// TwinCAT 3 PLC project Main
// ProgramVersion: 3.1.4023.0
// libraries:
//   Tc2_ModbusSrv, * (Beckhoff Automation GmbH)
//   Tc2_Standard, * (Beckhoff Automation GmbH)
//   Tc2_System, * (Beckhoff Automation GmbH)
//   Tc3_Module, * (Beckhoff Automation GmbH)
// project tree:
//   GVLs/ gvl_ha.TcGVL, gvl_mb.TcGVL, gvl_EA.TcGVL, gvl_RETAIN.TcGVL
//   / PLC1_Main.TcTTO
//   POUs/FB/ FB_Convert_2co2.TcPOU, FB_Convert_2temp.TcPOU, FB_Convert_2Zisterne.TcPOU, FB_Con_2_Value.TcPOU, FB_Count.TcPOU, FB_GarageStatus.TcPOU, FB_Heating.TcPOU, FB_Door.TcPOU, FB_Impulse_LongPress.TcPOU, FB_Light.TcPOU, FB_Impulse.TcPOU, FB_LightDimm.TcPOU, FB_LightDimmIndirectNC.TcPOU, FB_LightPIR.TcPOU, FB_ArithMittel10.TcPOU, FB_PowerSocket.TcPOU, FB_Fan.TcPOU, TP_RST.TcPOU
//   POUs/Light/ F_DimmAlgoForSwitch.TcPOU, F_LightDimmingConvertForHA.TcPOU
//   POUs/ MAIN.TcPOU, sub_Heating.TcPOU, sub_Light.TcPOU, sub_Access.TcPOU, sub_Measure.TcPOU, sub_Security.TcPOU, sub_Power.TcPOU
// real-time tasks:
//   TASK PLC1_Main: cycle T#10ms, priority 1, ADS port 350
// I/O:
//   DEVICE Gerät 1 (Beckhoff CCAT)
//   DEVICE CX8190
//     Schaltschrank (CX8190)
//   DEVICE Virtual-Ethernet
//     Werkstatt (BK9000)
// variable links:
//   Main/Main Instance <-> CX8190/Schaltschrank (CX8190)
//     PLC1_Main Inputs/gvl_EA.bID01_1 <-> ID01 (KL1104)/Channel 1/Eingang
//     PLC1_Main Inputs/gvl_EA.bID01_2 <-> ID01 (KL1104)/Channel 2/Eingang
//     PLC1_Main Inputs/gvl_EA.bID01_3 <-> ID01 (KL1104)/Channel 3/Eingang
//     PLC1_Main Inputs/gvl_EA.bID01_4 <-> ID01 (KL1104)/Channel 4/Eingang
//     PLC1_Main Inputs/gvl_EA.bID02_1 <-> ID02 (KL1104)/Channel 1/Eingang
//     PLC1_Main Inputs/gvl_EA.bID02_2 <-> ID02 (KL1104)/Channel 2/Eingang
//     PLC1_Main Inputs/gvl_EA.bID02_3 <-> ID02 (KL1104)/Channel 3/Eingang
//     PLC1_Main Inputs/gvl_EA.bID02_4 <-> ID02 (KL1104)/Channel 4/Eingang
//     PLC1_Main Inputs/gvl_EA.bID03_1 <-> ID03 (KL1104)/Channel 1/Eingang
//     PLC1_Main Inputs/gvl_EA.bID03_2 <-> ID03 (KL1104)/Channel 2/Eingang
//     PLC1_Main Inputs/gvl_EA.bID03_3 <-> ID03 (KL1104)/Channel 3/Eingang
//     PLC1_Main Inputs/gvl_EA.bID03_4 <-> ID03 (KL1104)/Channel 4/Eingang
//     PLC1_Main Inputs/gvl_EA.bID04_1 <-> ID04 (KL1104)/Channel 1/Eingang
//     PLC1_Main Inputs/gvl_EA.bID04_2 <-> ID04 (KL1104)/Channel 2/Eingang
//     PLC1_Main Inputs/gvl_EA.bID04_3 <-> ID04 (KL1104)/Channel 3/Eingang
//     PLC1_Main Inputs/gvl_EA.bID04_4 <-> ID04 (KL1104)/Channel 4/Eingang
//     PLC1_Main Inputs/gvl_EA.bID05_1 <-> ID05 (KL1104)/Channel 1/Eingang
//     PLC1_Main Inputs/gvl_EA.bID05_2 <-> ID05 (KL1104)/Channel 2/Eingang
//     PLC1_Main Inputs/gvl_EA.bID05_3 <-> ID05 (KL1104)/Channel 3/Eingang
//     PLC1_Main Inputs/gvl_EA.bID05_4 <-> ID05 (KL1104)/Channel 4/Eingang
//     PLC1_Main Inputs/gvl_EA.bID06_1 <-> ID06 (KL1104)/Channel 1/Eingang
//     PLC1_Main Inputs/gvl_EA.bID06_2 <-> ID06 (KL1104)/Channel 2/Eingang
//     PLC1_Main Inputs/gvl_EA.bID06_3 <-> ID06 (KL1104)/Channel 3/Eingang
//     PLC1_Main Inputs/gvl_EA.bID06_4 <-> ID06 (KL1104)/Channel 4/Eingang
//     PLC1_Main Inputs/gvl_EA.bID24_01_1 <-> ID24-01 (KL1104)/Channel 1/Eingang
//     PLC1_Main Inputs/gvl_EA.bID24_01_2 <-> ID24-01 (KL1104)/Channel 2/Eingang
//     PLC1_Main Inputs/gvl_EA.bID24_01_3 <-> ID24-01 (KL1104)/Channel 3/Eingang
//     PLC1_Main Inputs/gvl_EA.bID24_01_4 <-> ID24-01 (KL1104)/Channel 4/Eingang
//     PLC1_Main Inputs/gvl_EA.bID24_02_1 <-> ID24-02 (KL1104)/Channel 1/Eingang
//     PLC1_Main Inputs/gvl_EA.bID24_02_2 <-> ID24-02 (KL1104)/Channel 2/Eingang
//     PLC1_Main Inputs/gvl_EA.bID24_02_3 <-> ID24-02 (KL1104)/Channel 3/Eingang
//     PLC1_Main Inputs/gvl_EA.bID24_02_4 <-> ID24-02 (KL1104)/Channel 4/Eingang
//     PLC1_Main Inputs/gvl_EA.bID24_03_1 <-> ID24-03 (KL1104)/Channel 1/Eingang
//     PLC1_Main Inputs/gvl_EA.bID24_03_2 <-> ID24-03 (KL1104)/Channel 2/Eingang
//     PLC1_Main Inputs/gvl_EA.bID24_03_3 <-> ID24-03 (KL1104)/Channel 3/Eingang
//     PLC1_Main Inputs/gvl_EA.bID24_03_4 <-> ID24-03 (KL1104)/Channel 4/Eingang
//     PLC1_Main Inputs/gvl_EA.iIAA01_1 <-> IAA01 (KL3022)/Channel 1/Daten Ein
//     PLC1_Main Inputs/gvl_EA.iIAPT_01_1 <-> IAPT_01 (KL3214)/Channel 1/Daten Ein
//     PLC1_Main Inputs/gvl_EA.iIAV01_1 <-> IAV01 (KL3064)/Channel 1/Daten Ein
//     PLC1_Main Inputs/gvl_EA.iIAV01_2 <-> IAV01 (KL3064)/Channel 2/Daten Ein
//     PLC1_Main Inputs/gvl_EA.iIAV01_3 <-> IAV01 (KL3064)/Channel 3/Daten Ein
//     PLC1_Main Inputs/gvl_EA.iIAV01_4 <-> IAV01 (KL3064)/Channel 4/Daten Ein
//     PLC1_Main Inputs/gvl_EA.iIAV02_1 <-> IAV02 (KL3064)/Channel 1/Daten Ein
//     PLC1_Main Inputs/gvl_EA.iIAV02_2 <-> IAV02 (KL3064)/Channel 2/Daten Ein
//     PLC1_Main Inputs/gvl_EA.iIAV02_3 <-> IAV02 (KL3064)/Channel 3/Daten Ein
//     PLC1_Main Inputs/gvl_EA.iIAV02_4 <-> IAV02 (KL3064)/Channel 4/Daten Ein
//     PLC1_Main Outputs/gvl_EA.bOD01_1 <-> OD01 (KL2408)/Channel 1/Ausgang
//     PLC1_Main Outputs/gvl_EA.bOD01_2 <-> OD01 (KL2408)/Channel 2/Ausgang
//     PLC1_Main Outputs/gvl_EA.bOD01_3 <-> OD01 (KL2408)/Channel 3/Ausgang
//     PLC1_Main Outputs/gvl_EA.bOD01_4 <-> OD01 (KL2408)/Channel 4/Ausgang
//     PLC1_Main Outputs/gvl_EA.bOD01_5 <-> OD01 (KL2408)/Channel 5/Ausgang
//     PLC1_Main Outputs/gvl_EA.bOD01_6 <-> OD01 (KL2408)/Channel 6/Ausgang
//     PLC1_Main Outputs/gvl_EA.bOD01_7 <-> OD01 (KL2408)/Channel 7/Ausgang
//     PLC1_Main Outputs/gvl_EA.bOD01_8 <-> OD01 (KL2408)/Channel 8/Ausgang
//     PLC1_Main Outputs/gvl_EA.bOD02_1 <-> OD02 (KL2408)/Channel 1/Ausgang
//     PLC1_Main Outputs/gvl_EA.bOD02_2 <-> OD02 (KL2408)/Channel 2/Ausgang
//     PLC1_Main Outputs/gvl_EA.bOD02_3 <-> OD02 (KL2408)/Channel 3/Ausgang
//     PLC1_Main Outputs/gvl_EA.bOD02_4 <-> OD02 (KL2408)/Channel 4/Ausgang
//     PLC1_Main Outputs/gvl_EA.bOD02_5 <-> OD02 (KL2408)/Channel 5/Ausgang
//     PLC1_Main Outputs/gvl_EA.bOD02_6 <-> OD02 (KL2408)/Channel 6/Ausgang
//     PLC1_Main Outputs/gvl_EA.bOD02_7 <-> OD02 (KL2408)/Channel 7/Ausgang
//     PLC1_Main Outputs/gvl_EA.bOD02_8 <-> OD02 (KL2408)/Channel 8/Ausgang
//     PLC1_Main Outputs/gvl_EA.bOD03_1 <-> OD03 (KL2408)/Channel 1/Ausgang
//     PLC1_Main Outputs/gvl_EA.bOD03_2 <-> OD03 (KL2408)/Channel 2/Ausgang
//     PLC1_Main Outputs/gvl_EA.bOD03_3 <-> OD03 (KL2408)/Channel 3/Ausgang
//     PLC1_Main Outputs/gvl_EA.bOD03_4 <-> OD03 (KL2408)/Channel 4/Ausgang
//     PLC1_Main Outputs/gvl_EA.bOD03_5 <-> OD03 (KL2408)/Channel 5/Ausgang
//     PLC1_Main Outputs/gvl_EA.bOD03_6 <-> OD03 (KL2408)/Channel 6/Ausgang
//     PLC1_Main Outputs/gvl_EA.bOD03_7 <-> OD03 (KL2408)/Channel 7/Ausgang
//     PLC1_Main Outputs/gvl_EA.bOD03_8 <-> OD03 (KL2408)/Channel 8/Ausgang
//     PLC1_Main Outputs/gvl_EA.bOD04_1 <-> OD04 (KL2408)/Channel 1/Ausgang
//     PLC1_Main Outputs/gvl_EA.bOD04_2 <-> OD04 (KL2408)/Channel 2/Ausgang
//     PLC1_Main Outputs/gvl_EA.bOD04_3 <-> OD04 (KL2408)/Channel 3/Ausgang
//     PLC1_Main Outputs/gvl_EA.bOD04_4 <-> OD04 (KL2408)/Channel 4/Ausgang
//     PLC1_Main Outputs/gvl_EA.bOD04_5 <-> OD04 (KL2408)/Channel 5/Ausgang
//     PLC1_Main Outputs/gvl_EA.bOD04_6 <-> OD04 (KL2408)/Channel 6/Ausgang
//     PLC1_Main Outputs/gvl_EA.bOD04_7 <-> OD04 (KL2408)/Channel 7/Ausgang
//     PLC1_Main Outputs/gvl_EA.bOD04_8 <-> OD04 (KL2408)/Channel 8/Ausgang
//     PLC1_Main Outputs/gvl_EA.iOA01_1 <-> OA01 (KL4004)/Channel 1/Daten Aus
//     PLC1_Main Outputs/gvl_EA.iOA01_2 <-> OA01 (KL4004)/Channel 2/Daten Aus
//     PLC1_Main Outputs/gvl_EA.iOA01_3 <-> OA01 (KL4004)/Channel 3/Daten Aus
//     PLC1_Main Outputs/gvl_EA.iOA01_4 <-> OA01 (KL4004)/Channel 4/Daten Aus
//     PLC1_Main Outputs/gvl_EA.iOADim01 <-> OADim01 (KL2751)/Channel 1/Daten Aus
//     PLC1_Main Outputs/gvl_EA.iOADim02 <-> OADim02 (KL2751)/Channel 1/Daten Aus
//   Main/Main Instance <-> Virtual-Ethernet/Werkstatt (BK9000)
//     PLC1_Main Inputs/gvl_EA.bWID01_1 <-> bWID01 (KL1809)/Channel 1/Eingang
//     PLC1_Main Inputs/gvl_EA.bWID01_10 <-> bWID01 (KL1809)/Channel 10/Eingang
//     PLC1_Main Inputs/gvl_EA.bWID01_11 <-> bWID01 (KL1809)/Channel 11/Eingang
//     PLC1_Main Inputs/gvl_EA.bWID01_12 <-> bWID01 (KL1809)/Channel 12/Eingang
//     PLC1_Main Inputs/gvl_EA.bWID01_13 <-> bWID01 (KL1809)/Channel 13/Eingang
//     PLC1_Main Inputs/gvl_EA.bWID01_14 <-> bWID01 (KL1809)/Channel 14/Eingang
//     PLC1_Main Inputs/gvl_EA.bWID01_15 <-> bWID01 (KL1809)/Channel 15/Eingang
//     PLC1_Main Inputs/gvl_EA.bWID01_16 <-> bWID01 (KL1809)/Channel 16/Eingang
//     PLC1_Main Inputs/gvl_EA.bWID01_2 <-> bWID01 (KL1809)/Channel 2/Eingang
//     PLC1_Main Inputs/gvl_EA.bWID01_3 <-> bWID01 (KL1809)/Channel 3/Eingang
//     PLC1_Main Inputs/gvl_EA.bWID01_4 <-> bWID01 (KL1809)/Channel 4/Eingang
//     PLC1_Main Inputs/gvl_EA.bWID01_5 <-> bWID01 (KL1809)/Channel 5/Eingang
//     PLC1_Main Inputs/gvl_EA.bWID01_6 <-> bWID01 (KL1809)/Channel 6/Eingang
//     PLC1_Main Inputs/gvl_EA.bWID01_7 <-> bWID01 (KL1809)/Channel 7/Eingang
//     PLC1_Main Inputs/gvl_EA.bWID01_8 <-> bWID01 (KL1809)/Channel 8/Eingang
//     PLC1_Main Inputs/gvl_EA.bWID01_9 <-> bWID01 (KL1809)/Channel 9/Eingang
//     PLC1_Main Inputs/gvl_EA.bWID02_1 <-> bWID02 (KL1809)/Channel 1/Eingang
//     PLC1_Main Inputs/gvl_EA.bWID02_10 <-> bWID02 (KL1809)/Channel 10/Eingang
//     PLC1_Main Inputs/gvl_EA.bWID02_11 <-> bWID02 (KL1809)/Channel 11/Eingang
//     PLC1_Main Inputs/gvl_EA.bWID02_12 <-> bWID02 (KL1809)/Channel 12/Eingang
//     PLC1_Main Inputs/gvl_EA.bWID02_13 <-> bWID02 (KL1809)/Channel 13/Eingang
//     PLC1_Main Inputs/gvl_EA.bWID02_14 <-> bWID02 (KL1809)/Channel 14/Eingang
//     PLC1_Main Inputs/gvl_EA.bWID02_15 <-> bWID02 (KL1809)/Channel 15/Eingang
//     PLC1_Main Inputs/gvl_EA.bWID02_16 <-> bWID02 (KL1809)/Channel 16/Eingang
//     PLC1_Main Inputs/gvl_EA.bWID02_2 <-> bWID02 (KL1809)/Channel 2/Eingang
//     PLC1_Main Inputs/gvl_EA.bWID02_3 <-> bWID02 (KL1809)/Channel 3/Eingang
//     PLC1_Main Inputs/gvl_EA.bWID02_4 <-> bWID02 (KL1809)/Channel 4/Eingang
//     PLC1_Main Inputs/gvl_EA.bWID02_5 <-> bWID02 (KL1809)/Channel 5/Eingang
//     PLC1_Main Inputs/gvl_EA.bWID02_6 <-> bWID02 (KL1809)/Channel 6/Eingang
//     PLC1_Main Inputs/gvl_EA.bWID02_7 <-> bWID02 (KL1809)/Channel 7/Eingang
//     PLC1_Main Inputs/gvl_EA.bWID02_8 <-> bWID02 (KL1809)/Channel 8/Eingang
//     PLC1_Main Inputs/gvl_EA.bWID02_9 <-> bWID02 (KL1809)/Channel 9/Eingang
//     PLC1_Main Inputs/gvl_EA.iWIAA01_1 <-> IWAA01 (KL3022)/Channel 1/Daten Ein
//     PLC1_Main Inputs/gvl_EA.iWIAA01_2 <-> IWAA01 (KL3022)/Channel 2/Daten Ein
//     PLC1_Main Inputs/gvl_EA.iWIAA02_1 <-> IWAA02 (KL3054)/Channel 1/Daten Ein
//     PLC1_Main Inputs/gvl_EA.iWIAA02_2 <-> IWAA02 (KL3054)/Channel 2/Daten Ein
//     PLC1_Main Inputs/gvl_EA.iWIAA02_3 <-> IWAA02 (KL3054)/Channel 3/Daten Ein
//     PLC1_Main Inputs/gvl_EA.iWIAA02_4 <-> IWAA02 (KL3054)/Channel 4/Daten Ein
//     PLC1_Main Inputs/gvl_EA.iWIAV01_1 <-> IWAV01 (KL3064)/Channel 1/Daten Ein
//     PLC1_Main Inputs/gvl_EA.iWIAV01_2 <-> IWAV01 (KL3064)/Channel 2/Daten Ein
//     PLC1_Main Inputs/gvl_EA.iWIAV01_3 <-> IWAV01 (KL3064)/Channel 3/Daten Ein
//     PLC1_Main Inputs/gvl_EA.iWIAV01_4 <-> IWAV01 (KL3064)/Channel 4/Daten Ein
//     PLC1_Main Outputs/gvl_EA.bWOD01_1 <-> bWOD01 (KL2809)/Channel 1/Ausgang
//     PLC1_Main Outputs/gvl_EA.bWOD01_10 <-> bWOD01 (KL2809)/Channel 10/Ausgang
//     PLC1_Main Outputs/gvl_EA.bWOD01_11 <-> bWOD01 (KL2809)/Channel 11/Ausgang
//     PLC1_Main Outputs/gvl_EA.bWOD01_12 <-> bWOD01 (KL2809)/Channel 12/Ausgang
//     PLC1_Main Outputs/gvl_EA.bWOD01_13 <-> bWOD01 (KL2809)/Channel 13/Ausgang
//     PLC1_Main Outputs/gvl_EA.bWOD01_14 <-> bWOD01 (KL2809)/Channel 14/Ausgang
//     PLC1_Main Outputs/gvl_EA.bWOD01_15 <-> bWOD01 (KL2809)/Channel 15/Ausgang
//     PLC1_Main Outputs/gvl_EA.bWOD01_16 <-> bWOD01 (KL2809)/Channel 16/Ausgang
//     PLC1_Main Outputs/gvl_EA.bWOD01_2 <-> bWOD01 (KL2809)/Channel 2/Ausgang
//     PLC1_Main Outputs/gvl_EA.bWOD01_3 <-> bWOD01 (KL2809)/Channel 3/Ausgang
//     PLC1_Main Outputs/gvl_EA.bWOD01_4 <-> bWOD01 (KL2809)/Channel 4/Ausgang
//     PLC1_Main Outputs/gvl_EA.bWOD01_5 <-> bWOD01 (KL2809)/Channel 5/Ausgang
//     PLC1_Main Outputs/gvl_EA.bWOD01_6 <-> bWOD01 (KL2809)/Channel 6/Ausgang
//     PLC1_Main Outputs/gvl_EA.bWOD01_7 <-> bWOD01 (KL2809)/Channel 7/Ausgang
//     PLC1_Main Outputs/gvl_EA.bWOD01_8 <-> bWOD01 (KL2809)/Channel 8/Ausgang
//     PLC1_Main Outputs/gvl_EA.bWOD01_9 <-> bWOD01 (KL2809)/Channel 9/Ausgang
//     PLC1_Main Outputs/gvl_EA.bWOD02_1 <-> bWOD02 (KL2809)/Channel 1/Ausgang
//     PLC1_Main Outputs/gvl_EA.bWOD02_10 <-> bWOD02 (KL2809)/Channel 10/Ausgang
//     PLC1_Main Outputs/gvl_EA.bWOD02_11 <-> bWOD02 (KL2809)/Channel 11/Ausgang
//     PLC1_Main Outputs/gvl_EA.bWOD02_12 <-> bWOD02 (KL2809)/Channel 12/Ausgang
//     PLC1_Main Outputs/gvl_EA.bWOD02_13 <-> bWOD02 (KL2809)/Channel 13/Ausgang
//     PLC1_Main Outputs/gvl_EA.bWOD02_14 <-> bWOD02 (KL2809)/Channel 14/Ausgang
//     PLC1_Main Outputs/gvl_EA.bWOD02_15 <-> bWOD02 (KL2809)/Channel 15/Ausgang
//     PLC1_Main Outputs/gvl_EA.bWOD02_16 <-> bWOD02 (KL2809)/Channel 16/Ausgang
//     PLC1_Main Outputs/gvl_EA.bWOD02_2 <-> bWOD02 (KL2809)/Channel 2/Ausgang
//     PLC1_Main Outputs/gvl_EA.bWOD02_3 <-> bWOD02 (KL2809)/Channel 3/Ausgang
//     PLC1_Main Outputs/gvl_EA.bWOD02_4 <-> bWOD02 (KL2809)/Channel 4/Ausgang
//     PLC1_Main Outputs/gvl_EA.bWOD02_5 <-> bWOD02 (KL2809)/Channel 5/Ausgang
//     PLC1_Main Outputs/gvl_EA.bWOD02_6 <-> bWOD02 (KL2809)/Channel 6/Ausgang
//     PLC1_Main Outputs/gvl_EA.bWOD02_7 <-> bWOD02 (KL2809)/Channel 7/Ausgang
//     PLC1_Main Outputs/gvl_EA.bWOD02_8 <-> bWOD02 (KL2809)/Channel 8/Ausgang
//     PLC1_Main Outputs/gvl_EA.bWOD02_9 <-> bWOD02 (KL2809)/Channel 9/Ausgang

CONFIGURATION Main
    RESOURCE PLC ON TwinCAT3
        TASK PLC1_Main(INTERVAL := T#10ms, PRIORITY := 1);
        PROGRAM MAIN WITH PLC1_Main : MAIN;
    END_RESOURCE
END_CONFIGURATION

// ---- GVLs/gvl_ha.TcGVL
{attribute 'qualified_only'}
VAR_GLOBAL
	
//---------------WETTERSTATION-----------------------
	diWetterLUX			AT	%Q*:DINT;
	bWetterRAIN			AT	%Q*:BOOL;
	wWetterRAIN			AT	%Q*:WORD;
	diWetterWINDdir		AT	%Q*:DINT;
	diWetterWINDspeed	AT	%Q*:DINT;
	diWetterHUM			AT	%Q*:DINT;
	diWetterTEMP		AT	%Q*:DINT;	

END_VAR

// ---- GVLs/gvl_mb.TcGVL
{attribute 'qualified_only'}
VAR_GLOBAL
	
	Input_Coils        	: ARRAY [0..255] OF BOOL;  	//R/W BOOLS
	Input_Registers     : ARRAY [0..255] OF WORD;	//R/W 16-Bit Register
	
	Output_Coils	    : ARRAY [0..255] OF BOOL;	//Read Only BOOLS
	Output_Registers    : ARRAY [0..255] OF WORD;	//Read Only 16-Bit Register
	
END_VAR

(*-----------------------------------------------------------------------------
Output_Coils[0]		- 1000 <- Licht Küche
Output_Coils[1] 	- 1001 <- Licht Hausgang EG
Output_Coils[2] 	- 1002 <- Aussenbeleuchtung OST 		
Output_Coils[3] 	- 1003 <- Aussenbeleuchtung Haustür 	
Output_Coils[4] 	- 1004 <- Licht Technikraum
Output_Coils[5] 	- 1005 <- Licht Hobbyraum
Output_Coils[6] 	- 1006 <- Licht Werkstatt
Output_Coils[7] 	- 1007 <- Licht Esszimmertisch
Output_Coils[8] 	- 1008 <- Licht Esszimmer
Output_Coils[9] 	- 1009 <- Licht Wohnzimmer
Output_Coils[10] 	- 1010 <- Aussenbeleuchtung Balkon
Output_Coils[11] 	- 1011 <- Wohnzimmer Steckdose Uhr
Output_Coils[12] 	- 1012 <- Werkstatt Steckdose
Output_Coils[13] 	- 1013 <- Garagentor Stellung Toggle Impuls
Output_Coils[14] 	- 1014 <- Türgong Impuls
Output_Coils[15] 	- 1015 <- Vitramo Bad
Output_Coils[16] 	- 1016 <- Haustüröffner Impuls
Output_Coils[17] 	- 1017 <- Haustüröffner Dauer
Output_Coils[18] 	- 1018 <- Wohnzimmer Steckdose Fernseher
Output_Coils[19] 	- 1019 <- ENV_NoDailight
Output_Coils[20] 	- 1020 <- Wohnzimmer Steckdose Esszimmer
Output_Coils[21] 	- 1021 <- Aussensteckdose Haustür
Output_Coils[22] 	- 1022 <- Aussensteckdose Balkon
Output_Coils[23] 	- 1023 <- Strom Zisternenpumpe
Output_Coils[24] 	- 1024 <- Strom SmartMirror
Output_Coils[25] 	- 1025 <- Wohnzimmer Steckdose LED-Band
Output_Coils[26] 	- 1026 <- Lüfter Werkstatt
Output_Coils[27] 	- 1027 <- Strom Ladegeräte Werkstatt
Output_Coils[28] 	- 1028 <- Aussenbeleuchtung Treppe Süd
Output_Coils[29] 	- 1029 <- Eingang Bewegungsmelder Treppe Süd
Output_Coils[30] 	- 1030 <- Licht Garage
Output_Coils[31] 	- 1031 <- Eingang Bewegungsmelder Überdachung OST
Output_Coils[32] 	- 1032 <- Licht Aussen Hauseingang
Output_Coils[33] 	- 1033 <- Ventilator Garage
Output_Coils[34] 	- 1034 <- Türöffner  Garage Strasse
Output_Coils[35] 	- 1035 <- Türöffner Garage Haus
Output_Coils[36] 	- 1036 <- Garagentormotor Licht AN / AUS
Output_Coils[37] 	- 1037 <- Garagentor Stellung Lüften impuls
Output_Coils[38] 	- 1038 <- Garagentor Stellung AUF impuls
Output_Coils[39] 	- 1039 <- Garagentor Stellung AB impuls
Output_Coils[40] 	- 1040 <- Garagentor Stellung 1/2 impuls
Output_Coils[41] 	- 1041 <- Türöffner Werkstatt
Output_Coils[42] 	- 1042 <- Entfeuchter Werkstatt
Output_Coils[43] 	- 1043 <- Strom Ladegeräte Garage
Output_Coils[44] 	- 1044 <- Steckdose Garagendach

########################----FENSTER / TÜRKONTAKTE----################
Output_coils[200]	- 1200 <- Fenster 	EG 	BAD
Output_coils[201]	- 1201 <- Fenster 	EG 	Büro
Output_coils[202]	- 1202 <- Tür		EG	Balkontür
Output_coils[203]	- 1203 <- Fenster	UG	Keller
Output_coils[204]	- 1204 <- Fenster	UG	Technik
Output_coils[205]	- 1205 <- Fenster	UG	Hobbyraum Süd
Output_coils[206]	- 1206 <- Fenster	UG	Hobbyraum West
Output_coils[207]	- 1207 <- Tür		UG	Terassentür
Output_coils[208]	- 1208 <- Fenster	UG	Werkstatt
Output_coils[209]	- 1209 <- Tür		UG	Werkstatt
Output_coils[210]	- 1210 <- Tür		OG	Garage Strasse
Output_coils[211]	- 1211 <- Fenster	OG	Garage
Output_coils[212]	- 1212 <- Tür		OG	Garage Haus
Output_coils[213]	- 1213 <- Garagentor Status offen
Output_coils[214]	- 1214 <- Garagentor Status geschlossen
Output_coils[215]	- 1215 <- Garagentor Status Lüftung




########################----ALARM----################################
Output_coils[240]	- 1240 <- Aktiviert alle Alarmfunktionen

Output_coils[241]	- 1241 <- Aktiviert dauerhaft alle Lichter
Output_coils[242]	- 1242 <- Aktiviert dauerhaft alle Lichter INNEN
Output_coils[243]	- 1243 <- Aktiviert dauerhaft alle Lichter AUSSEN

Output_coils[244]	- 1244 <- Aktiviert dauerhaft alle Alarmsignale
Output_coils[245]	- 1245 <- Aktiviert dauerhaft alle Alarmsignale INNEN
Output_coils[246]	- 1246 <- Aktiviert dauerhaft alle Alarmsignale AUSSEN

Output_coils[247]	- 1247 <- 
Output_coils[248]	- 1248 <- 
Output_coils[249]	- 1249 <- 
Output_coils[250]	- 1250 <- 

Output_coils[251]	- 1251 <- Aktiviert Testalarm Esszimmertisch
Output_coils[252]	- 1252 <- Aktiviert Testalarm Esszimmer
Output_coils[253]	- 1253 <- Aktiviert Testalarm Wohnzimmer
Output_coils[254]	- 1254 <- Aktiviert Testalarm Balkon
Output_coils[255]	- 1255 <- 



------------------------------------------------------------------------------*)

(*-----------------------------------------------------------------------------
Output_Registers[0] 	- 2000 <- Trinkwasserverbrauch gvl_RETAIN 
Output_Registers[7] 	- 2007 <- Helligkeit Esszimmertisch
Output_Registers[8] 	- 2008 <- Helligkeit Esszimmer
Output_Registers[9] 	- 2009 <- Helligkeit Wohnzimmer
Output_Registers[10] 	- 2010 <- Helligkeit Aussenbeleuchtung Balkon
Output_Registers[11] 	- 2011 <- 
Output_Registers[12] 	- 2012 <- Zisterne Füllstand Prozent
Output_Registers[13] 	- 2013 <- Zisterne Füllstand Liter
Output_Registers[14] 	- 2014 <- Wohnzimmer Temperatur
Output_Registers[15] 	- 2015 <- Wohnzimmer Feuchtigkeit
Output_Registers[16] 	- 2016 <- Wohnzimmer CO2
Output_Registers[17] 	- 2017 <- Technikraum Temperatur
Output_Registers[18] 	- 2018 <- Technikraum Feuchtigkeit
Output_Registers[19] 	- 2019 <- Dachboden Temperatur
Output_Registers[20] 	- 2020 <- Werkstatt Temperatur
Output_Registers[21] 	- 2021 <- Werkstatt Feuchtigkeit
Output_Registers[22] 	- 2022 <- Zisternenwasserverbrauch gvl_RETAIN
Output_Registers[23] 	- 2023 <- Garage Temperatur
Output_Registers[24] 	- 2024 <- Garage Feuchtigkeit
Output_Registers[25] 	- 2025 <- Status Garagentor
Output_Registers[26] 	- 2026 <- AUSSEN Temperatur
Output_Registers[27] 	- 2027 <- AUSSEN relative Feuchte (%)
Output_Registers[28] 	- 2028 <- AUSSEN Regenmenge in mm (gvl_Retaun)
Output_Registers[29] 	- 2029 <- AUSSEN Windgeschwindigkeit m/s
Output_Registers[30] 	- 2030 <- AUSSEN Windgeschwindigkeit km/h
Output_Registers[31] 	- 2031 <- AUSSEN Windrichtung Grad




------------------------------------------------------------------------------*)

// ---- GVLs/gvl_EA.TcGVL
VAR_GLOBAL
	(* -------------------------------------------------------------------
	Beispielvariablendeklaration (%Q* = Ausgang; %I* = Eingang:
	bAusgang1			AT %Q*:BOOL;
	abAusgaenge			AT %Q*:ARRAY[0..7] OF BOOL;
	bEingang			AT %I*:BOOL;
	iSollwertAnalog  	AT %Q*:INT;
	
	Nach deklaration muss das Projekt neu Erstellt werden und die Konfiguration aktiviert werden.
	Dann kann bei den E/A Geräten die Zuordnung der Variable zum Eingang / Ausgang gemacht werden.
	
	INFO:
	im HASS muss die Variable mit .bAusgang angesprochen werden.
	---------------------------------------------------------------------- *)
	
	//----------OD01----------------------
	bOD01_1		AT	%Q*:BOOL;
	bOD01_2		AT	%Q*:BOOL;			// Lampe L2 Indirekt (Esszimmer) ACHTUNG NC
	bOD01_3		AT	%Q*:BOOL;			// Lampe L3 Indirekt (Wohnzimmer)
	bOD01_4		AT	%Q*:BOOL;			// Lampe L4 (Küche)
	bOD01_5		AT	%Q*:BOOL;			// Lampe L5 (Diele EG)
	bOD01_6		AT	%Q*:BOOL;			// Aussenlampe L6 (OST Rechts von Haustür)
	bOD01_7		AT	%Q*:BOOL;			// Aussenlampe L7 (OST Links von Haustür)
	bOD01_8		AT	%Q*:BOOL;			// Aussenlampe L8 (Süd - Ost)
	
	//----------OD02----------------------
	bOD02_1		AT	%Q*:BOOL;			// Aussenlampe L9 (Balkon Rechts)
	bOD02_2		AT	%Q*:BOOL;			// Aussenlampe L10 (Balkon Links)
	bOD02_3		AT	%Q*:BOOL;			// Tür-Gong
	bOD02_4		AT	%Q*:BOOL := TRUE;	// Steckdose S1 (Ecke Esszimmer SW)
	bOD02_5		AT	%Q*:BOOL := TRUE;	// Steckdose S2 (Balkontür Rechts Esszimmer)
	bOD02_6		AT	%Q*:BOOL;			// Steckdose S3 (Ecke Whonzimmer NW - Fernseher) ACHTUNG NC
	bOD02_7		AT	%Q*:BOOL;			// Aussensteckdose S4 (Haustür Rechts) 
	bOD02_8		AT	%Q*:BOOL;			// Aussensteckdose S5 (Balkon)

	//----------OD03----------------------
	bOD03_1		AT	%Q*:BOOL;			// Licht Hobbyraum Groß
	bOD03_2		AT	%Q*:BOOL;			// Licht Hobbyraum Klein
	bOD03_3		AT	%Q*:BOOL;			// Aussenlampe Süd-West
	bOD03_4		AT	%Q*:BOOL;			// Aussensteckdose Süd-West
	bOD03_5		AT	%Q*:BOOL;			// Licht Technikraum ACHTUNG NC
	bOD03_6		AT	%Q*:BOOL := TRUE;	// Zuleitung Strom Zisterne
	bOD03_7		AT	%Q*:BOOL;			// Aussenlampe West
	bOD03_8		AT	%Q*:BOOL;			// Aussensteckdose West

	//----------OD04----------------------
	bOD04_1		AT	%Q*:BOOL;			// Spot Küche
	bOD04_2		AT	%Q*:BOOL := TRUE;	// Zuleitung Niesche Diele EG
	bOD04_3		AT	%Q*:BOOL;			// Zuleitung Steckdose Lichtband
	bOD04_4		AT	%Q*:BOOL;			// Vitramo Bad OG
	bOD04_5		AT	%Q*:BOOL;			// Türöffner Haustür
	bOD04_6		AT	%Q*:BOOL;			//
	bOD04_7		AT	%Q*:BOOL;			//
	bOD04_8		AT	%Q*:BOOL;			//

	//----------OA01----------------------
	iOA01_1		AT	%Q*:INT;			//Wohnzimmer	0-10V Dimmer
	iOA01_2		AT	%Q*:INT;			//Esszimmer		0-10V Dimmer
	iOA01_3		AT	%Q*:INT;
	iOA01_4		AT	%Q*:INT;

	//----------ID01----------------------
	bID01_1		AT	%I*:BOOL; 			// 105 T1 (Esszimmer Indirekt)
	bID01_2		AT	%I*:BOOL; 			// 105 T2 (Wohnzimmer Indirekt)
	bID01_3		AT	%I*:BOOL; 			// 105 T3 (Deckenlampe Esstisch)
	bID01_4		AT	%I*:BOOL; 			// 104 T1 (Deckenlampe Küche)

	//----------ID02----------------------
	bID02_1		AT	%I*:BOOL;			// 105 T5 (Balkontür oben)
	bID02_2		AT	%I*:BOOL;			// 105 T6 (Balkontür unten)
	bID02_3		AT	%I*:BOOL;			// 115 T9 (Treppenabgang EG Oben)
	bID02_4		AT	%I*:BOOL;			// 115 T10 (Diele - Eingang Büro)

	//----------ID03----------------------
	bID03_1		AT	%I*:BOOL;			// 115 T11 (Diele - Eingang Esszimmer unten)
	bID03_2		AT	%I*:BOOL;			// 115 T12 (Diele - Haustür / Bad EG)
	bID03_3		AT	%I*:BOOL;			// Schalter Technikraum
	bID03_4		AT	%I*:BOOL;			// Bewegungsmelder Aussen L8 (Treppe Süd)

	//----------ID04----------------------
	bID04_1		AT	%I*:BOOL;			// Schalter Hobbyraum
	bID04_2		AT	%I*:BOOL;
	bID04_3		AT	%I*:BOOL;
	bID04_4		AT	%I*:BOOL;			// Heizungssteuerung K9 -> Vitramo Bad OG

	//----------ID05----------------------
	bID05_1		AT	%I*:BOOL;			// Taster Hausgang Garagentor
	bID05_2		AT	%I*:BOOL;			// Taster Hausgang Garagentür
	bID05_3		AT	%I*:BOOL;
	bID05_4		AT	%I*:BOOL;

	//----------ID06----------------------
	bID06_1		AT	%I*:BOOL;
	bID06_2		AT	%I*:BOOL;
	bID06_3		AT	%I*:BOOL;
	bID06_4		AT	%I*:BOOL;
	
	//----------ID24-01--------------------
	bID24_01_1		AT	%I*:BOOL;	// Türklingel Doorbird Aussen (R1)
	bID24_01_2		AT	%I*:BOOL;	// Türklingel Doorbird Innen (R1)
	bID24_01_3		AT	%I*:BOOL;	// Fensterkontakt Bad EG
	bID24_01_4		AT	%I*:BOOL;	// Fensterkontakt Büro
	
	//----------ID24-02--------------------
	bID24_02_1		AT	%I*:BOOL;	// Fensterkontakt Keller
	bID24_02_2		AT	%I*:BOOL;	// Fensterkontakt Technik
	bID24_02_3		AT	%I*:BOOL;	// Fensterkontakt Hobbyraum Süd
	bID24_02_4		AT	%I*:BOOL;	// Kontakt Terassentür UG
	
	//----------ID24-03--------------------
	bID24_03_1		AT	%I*:BOOL;	// Fensterkontakt Hobbyraum West
	bID24_03_2		AT	%I*:BOOL;	// Türkontakt Balkontür EG
	bID24_03_3		AT	%I*:BOOL;	// Wasseruhr Trinkwasser 	Impuls = 10 Liter
	bID24_03_4		AT	%I*:BOOL;	// Wasseruhr Zisterne 		Impuls = 1 Liter
	
	//----------OADim01---------------------
	iOADim01		AT	%Q*:INT;	// Dimmer Esszimmerlampe
	
	//----------OADim02---------------------
	iOADim02 		AT 	%Q*:INT;	// Dimmer Balkon
	
	//----------IAV01-----------------------
	iIAV01_1		AT	%I*:INT;	// Temperatur Wohnzimmer (°C)
	iIAV01_2		AT	%I*:INT;	// Feuchtigkeit Wohnzimmer (%)
	iIAV01_3		AT	%I*:INT;	// CO2 Wohnzimmer (ppm)
	iIAV01_4		AT	%I*:INT;	// Temperatur Technikraum (°C)
	
	//----------IAV02-----------------------
	iIAV02_1		AT	%I*:INT;	// Feuchtigkeit Technikraum (%)
	iIAV02_2		AT	%I*:INT;
	iIAV02_3		AT	%I*:INT;
	iIAV02_4		AT	%I*:INT;
	
	//----------IAA01-----------------------
	iIAA01_1		AT	%I*:INT;	//Füllstand Zisterne 4-20mA
	
	//----------IAPT_01---------------------
	iIAPT_01_1		AT	%I*:INT;	//PT Temp Bühne
	
	
	//-------------WERKSTATT-----------------------------
	
	//----------bWOD01-----------------------------------
	bWOD01_1		AT	%Q*:BOOL;				// Licht Werkstatt ACHTUNG NC
	bWOD01_2		AT	%Q*:BOOL;				// Strom Werkstatt
	bWOD01_3		AT	%Q*:BOOL;				// Entfeuchter Werkstatt
	bWOD01_4		AT	%Q*:BOOL;				// Lüfter UG
	bWOD01_5		AT	%Q*:BOOL;				// Ladegeräte Werkstatt
	bWOD01_6		AT	%Q*:BOOL;				// Garagentor Stellung Toggle
	bWOD01_7		AT	%Q*:BOOL;				// Licht Garage
	bWOD01_8		AT	%Q*:BOOL;				// Licht Überdachung
	bWOD01_9		AT	%Q*:BOOL;				// Ventilator Garage
	bWOD01_10		AT	%Q*:BOOL;				// Türöffner Garage Strasse
	bWOD01_11		AT	%Q*:BOOL;				// Türöffner Garage Haus
	bWOD01_12		AT	%Q*:BOOL;				// Garagentormotor Licht AN / AUS
	bWOD01_13		AT	%Q*:BOOL;				// Garagentor Stellung Lüften
	bWOD01_14		AT	%Q*:BOOL;				// Garagentor Stellung AUF
	bWOD01_15		AT	%Q*:BOOL;				// Garagentor Stellung AB
	bWOD01_16		AT	%Q*:BOOL;				// Garagentor Stellung 1/2
	
	//----------bWOD02-----------------------------------
	bWOD02_1		AT	%Q*:BOOL;				// Türöffner Werkstatt-Tür
	bWOD02_2		AT	%Q*:BOOL;				// Ladegeräte Garage
	bWOD02_3		AT	%Q*:BOOL;				// Steckdose Garagendach
	bWOD02_4		AT	%Q*:BOOL;				// 
	bWOD02_5		AT	%Q*:BOOL;				// 
	bWOD02_6		AT	%Q*:BOOL;				// 
	bWOD02_7		AT	%Q*:BOOL;				// 
	bWOD02_8		AT	%Q*:BOOL;				// 
	bWOD02_9		AT	%Q*:BOOL;				// 
	bWOD02_10		AT	%Q*:BOOL;				// 
	bWOD02_11		AT	%Q*:BOOL;				// 
	bWOD02_12		AT	%Q*:BOOL;				// 
	bWOD02_13		AT	%Q*:BOOL;				//
	bWOD02_14		AT	%Q*:BOOL;				// 
	bWOD02_15		AT	%Q*:BOOL;				// 
	bWOD02_16		AT	%Q*:BOOL;				//
	
	//---------bWID01-------------------------------------
	bWID01_1		AT	%I*:BOOL;				// LichtTaster Werksatt 
	bWID01_2		AT	%I*:BOOL;				// Stromschalter Werkstatt
	bWID01_3		AT	%I*:BOOL;				// Reedkontakt Werkstatttür
	bWID01_4		AT	%I*:BOOL;				// Reedkontakt Werkstattfenster
	bWID01_5		AT	%I*:BOOL;				// Taster Garage Haus
	bWID01_6		AT	%I*:BOOL;				// Taster Garage Strasse
	bWID01_7		AT	%I*:BOOL;				// Bewegungsmelder Überdachung
	bWID01_8		AT	%I*:BOOL;				// Garage Tür Strasse Input from Doorbird
	bWID01_9		AT	%I*:BOOL;				// Garage Tür Haus Input from Doorbird
	bWID01_10		AT	%I*:BOOL;				// Werkstatt Tür Input from Doorbird
	bWID01_11		AT	%I*:BOOL;				// Türkontakt Garagentür Strasse
	bWID01_12		AT	%I*:BOOL;				// Fensterkontakt Garage
	bWID01_13		AT	%I*:BOOL;				// Türkontakt Garagentür Haus
	bWID01_14		AT	%I*:BOOL;				// Lüftersignal Garagentorantrieb UAP1
	bWID01_15		AT	%I*:BOOL;				// Garagentor Status OFFEN
	bWID01_16		AT	%I*:BOOL;				// Garagentor Status GESCHLOSSEN
	
	//---------bWID02-------------------------------------
	bWID02_1		AT	%I*:BOOL;				// Licht Garagentor AN Rückmeldung
	bWID02_2		AT	%I*:BOOL;				// Regenmesser Garagendach Impuls = 0,3 mm Regen
	bWID02_3		AT	%I*:BOOL;				// Regenwächter
	bWID02_4		AT	%I*:BOOL;				// 
	bWID02_5		AT	%I*:BOOL;				// 
	bWID02_6		AT	%I*:BOOL;				// 
	bWID02_7		AT	%I*:BOOL;				// 
	bWID02_8		AT	%I*:BOOL;				// 
	bWID02_9		AT	%I*:BOOL;				// 
	bWID02_10		AT	%I*:BOOL;				// 
	bWID02_11		AT	%I*:BOOL;				// 
	bWID02_12		AT	%I*:BOOL;				// 
	bWID02_13		AT	%I*:BOOL;				// 
	bWID02_14		AT	%I*:BOOL;				// 
	bWID02_15		AT	%I*:BOOL;				// 
	bWID02_16		AT	%I*:BOOL;				// 
	
	//----------IWAV01-----------------------
	iWIAV01_1		AT	%I*:INT;	// Temperatur Werkstatt (-30 - +70 °C)
	iWIAV01_2		AT	%I*:INT;	// Feuchtigkeit Werkstatt (%)
	iWIAV01_3		AT	%I*:INT;	// Feuchtigkeit Garage (%)
	iWIAV01_4		AT	%I*:INT;	// Temperatur Garage (-30 - +70 °C)
	
	//----------IWAV01-----------------------
	iWIAA01_1		AT	%I*:INT;	// AUSSEN relative Feuchte
	iWIAA01_2		AT	%I*:INT;	// AUSSEN Temperatur (-30 - +70 °C)
	
		//----------IWAV01-----------------------
	iWIAA02_1		AT	%I*:INT;	// Windgeschwindigkeit max. 35m/s
	iWIAA02_2		AT	%I*:INT;	// Windrichtung
	iWIAA02_3		AT	%I*:INT;	// LUX aussenbereich
	iWIAA02_4		AT	%I*:INT;	//
	
END_VAR

// ---- GVLs/gvl_RETAIN.TcGVL
{attribute 'qualified_only'}
VAR_GLOBAL RETAIN
	//Brauchwassermenge verbraucht in m3
    waterConsumption : WORD;
	waterConsumptionZisterne : WORD;
	
	//Regenmenge in MM
	waterRain : WORD; 
END_VAR

// ---- POUs/MAIN.TcPOU
PROGRAM MAIN
VAR
END_VAR

//######################################################################################
//##------------------------------------ MAIN------- ---------------------------------##
//######################################################################################

sub_Light();
sub_Security();
sub_Access();
sub_Power();
sub_Measure();
sub_Heating();

END_PROGRAM

// ---- POUs/sub_Light.TcPOU
PROGRAM sub_Light
VAR
		fbLichtHausgang 		: FB_Light;
		fbLichtTechnikraum 		: FB_Light;
		fbLichtHobbyraum 		: FB_Light;
		fbLichtKueche			: FB_Light;
		fbLichtWerkstatt		: FB_Light;
		fbLichtGarage			: FB_Light;
		fbLichtEsstisch			: FB_LIghtDimm;
		fbLichtBalkon			: FB_LIghtDimm;
		fbLichtEsszimmer		: FB_LightDimmIndirectNC;
		fbLichtWohnzimmer		: FB_LightDimmIndirectNC;
		fbLichtAussenOST		: FB_LightPIR;
		fbLichtAussenHaustur	: FB_LightPIR;
		fbLichtAussenTreppeSud	: FB_LightPIR;
		fbLichtAussenEingang	: FB_LightPIR;
END_VAR

//###################################################################################
//##-----------------------------------BELEUCHTUNG---------------------------------##
//###################################################################################

//--------------------HAUSGANG EG----------------------------------
fbLichtHausgang.bInputs[0] 	:= gvl_EA.bID02_4;
fbLichtHausgang.bInputs[1] 	:= gvl_EA.bID03_1;
fbLichtHausgang.bInputs[2] 	:= gvl_EA.bID03_2;
fbLichtHausgang.bInputs[3] 	:= gvl_EA.bID02_3;

fbLichtHausgang.bInputsDoors[0] 	:= gvl_EA.bID24_01_2;

fbLichtHausgang
(
	bInputSec		:= gvl_mb.Output_Coils[242],
	bInputHA		:= gvl_mb.Output_Coils[1],
	bSunisDown		:= gvl_mb.Output_Coils[19],
	bOut 			=> gvl_EA.bOD01_5,
);
//-----------------------------------------------------------------

//--------------------KÜCHE----------------------------------------
fbLichtKueche.bInputs[0]	:= gvl_EA.bID01_4;

fbLichtKueche
(
	bInputSec	:= 	gvl_mb.Output_Coils[242],
	bInputHA	:=	gvl_mb.Output_Coils[0],
	bOut		=>	gvl_EA.bOD01_4, //Licht Küche
	bOut		=>	gvl_EA.bOD04_1,	//Spot Küche
);
//-----------------------------------------------------------------

//--------------------TECHNIKRAUM----------------------------------
fbLichtTechnikraum.bInputs[0] := gvl_EA.bID03_3;

fbLichtTechnikraum
(	
	bInputSec		:= gvl_mb.Output_Coils[242],
	bLightInv_NC	:= TRUE,
	bInputHA		:= gvl_mb.Output_Coils[4],
	bAllFlanks 		:= TRUE,
	bOut 			=> gvl_EA.bOD03_5,
);
//-----------------------------------------------------------------

//--------------------HOBBYRAUM------------------------------------
fbLichtHobbyraum.bInputs[0] := gvl_EA.bID04_1;

fbLichtHobbyraum
(	
	bInputSec		:= gvl_mb.Output_Coils[242],
	bInputHA		:= gvl_mb.Output_Coils[5],
	bAllFlanks 		:= TRUE,
	bOut 			=> gvl_EA.bOD03_1,
	bOut			=> gvl_EA.bOD03_2,
);
//-----------------------------------------------------------------

//--------------------WERKSTATT----------------------------------
fbLichtWerkstatt.bInputs[0] := gvl_EA.bWID01_1;

fbLichtWerkstatt.bInputsDoors[0] := gvl_mb.Output_coils[209];

fbLichtWerkstatt
(	
	bInputSec		:= gvl_mb.Output_Coils[242],
	bLightInv_NC	:= TRUE,
	bInputHA		:= gvl_mb.Output_Coils[6],
	bSunisDown		:= gvl_mb.Output_Coils[19],
	bOut 			=> gvl_EA.bWOD01_1,
);
//-----------------------------------------------------------------

//--------------------GARAGE----------------------------------
fbLichtGarage.bInputs[0] := gvl_EA.bWID01_5;
fbLichtGarage.bInputs[1] := gvl_EA.bWID01_6;

fbLichtGarage.bInputsDoors[0] := gvl_mb.Output_coils[210];
fbLichtGarage.bInputsDoors[1] := gvl_mb.Output_coils[212];

fbLichtGarage
(	
	bInputSec		:= gvl_mb.Output_Coils[242],
	bInputHA		:= gvl_mb.Output_Coils[30],
	bSunisDown		:= gvl_mb.Output_Coils[19],
	bOut 			=> gvl_EA.bWOD01_7,
);
//-----------------------------------------------------------------

//--------------------AUSSEN OST----------------------------------
fbLichtAussenOST
(	
	bInputSecLoop	:= gvl_mb.Output_Coils[243],
	bInputHA		:= gvl_mb.Output_Coils[2],
	bOut 			=> gvl_EA.bOD01_6,
);
//-----------------------------------------------------------------

//--------------------ESSTISCH----------------------------------
fbLichtEsstisch.bInputs[0] := gvl_EA.bID01_3;

fbLichtEsstisch
(	
	bInputSec		:= gvl_mb.Output_Coils[242],
	bInputSecTest	:= gvl_mb.Output_Coils[251],
	bInputHA		:= gvl_mb.Output_Coils[7],
	iDimmValue		:= gvl_mb.Output_Registers[7],
	iNumPress4Dimm	:= 4,
	iOut 			=> gvl_EA.iOADim01,
);
//-----------------------------------------------------------------

//--------------------BALKON----------------------------------
fbLichtBalkon.bInputs[0] := gvl_EA.bID02_2;

fbLichtBalkon
(	
	bInputSec		:= gvl_mb.Output_Coils[243],
	bInputSecTest	:= gvl_mb.Output_Coils[254],
	bInputHA		:= gvl_mb.Output_Coils[10],
	iDimmValue		:= gvl_mb.Output_Registers[10],
	bOnlyAtNight	:= TRUE,
	iNumPress4Dimm	:= 4,
	iOut 			=> gvl_EA.iOADim02,
);
//-----------------------------------------------------------------

//--------------------INDIREKTE BELEUCHTUNG ESSZIMMER--------------
fbLichtEsszimmer.bInputs[0] 	:= gvl_EA.bID01_1;
fbLichtEsszimmer.bInputs[1] 	:= gvl_EA.bID02_1;

fbLichtEsszimmer
(
	bInputSec		:= gvl_mb.Output_Coils[242],
	bInputSecTest	:= gvl_mb.Output_Coils[252],
	bInputHA		:= gvl_mb.Output_Coils[8],
	iDimmValue		:= gvl_mb.Output_Registers[8],
	iNumPress4Dimm	:= 4,
	iOut 			=> gvl_EA.iOA01_2,
	bOut			=> gvl_EA.bOD01_2,
);
//-----------------------------------------------------------------

//--------------------INDIREKTE BELEUCHTUNG WOHNZIMMER-------------
fbLichtWohnzimmer.bInputs[0] 	:= gvl_EA.bID01_2;

fbLichtWohnzimmer
(
	bInputSec		:= gvl_mb.Output_Coils[242],
	bInputSecTest	:= gvl_mb.Output_Coils[253],
	bInputHA		:= gvl_mb.Output_Coils[9],
	iDimmValue		:= gvl_mb.Output_Registers[9],
	iNumPress4Dimm	:= 4,
	iOut 			=> gvl_EA.iOA01_1,
	bOut			=> gvl_EA.bOD01_3,
);
//-----------------------------------------------------------------

//--------------------Aussenbeleuchtung Treppe Süd-------------
fbLichtAussenTreppeSud
(
	bInputSecLoop	:= gvl_mb.Output_Coils[243],
	bInputPIR		:= gvl_ea.bID03_4,
	bInputHA		:= gvl_mb.Output_Coils[28],
	tHigh			:= T#1M,
	bOut			=> gvl_ea.bOD01_8,
);

// Sync PIR to HA
gvl_mb.Output_Coils[29] := gvl_ea.bID03_4;
//-----------------------------------------------------------------

//--------------------Aussenbeleuchtung Eingang Haus-----------
fbLichtAussenEingang
(
	bInputSecLoop	:= gvl_mb.Output_Coils[243],
	bInputPIR		:= gvl_ea.bWID01_7,
	bInputHA		:= gvl_mb.Output_Coils[32],
	tHigh			:= T#1M,
	bOut			=> gvl_ea.bWOD01_8,
);

// Sync PIR to HA
gvl_mb.Output_Coils[31] := gvl_ea.bWID01_7;
//----------------------------------------------------------------

//--------------------AUSSEN HAUSTÜR----------------------------------
fbLichtAussenHaustur
(	
	bInputSecLoop	:= gvl_mb.Output_Coils[243],
	bInputPIR		:= gvl_ea.bWID01_7,
	tHigh			:= T#1M,
	bInputHA		:= gvl_mb.Output_Coils[3],
	bOut 			=> gvl_EA.bOD01_7,
);
//-----------------------------------------------------------------

END_PROGRAM

// ---- POUs/FB/FB_Light.TcPOU
FUNCTION_BLOCK FB_Light
VAR_INPUT
	bInputs			:	ARRAY[0..nSize] OF BOOL;	//Input Schalter oder Taster
	bInputsDoors	:	ARRAY[0..nSize] OF BOOL;	//Inputs for Door Contacts to put on light at Night
	bInputSec		:	BOOL := FALSE;				//Input für Security Schaltung
	bLightInv_NC	:	BOOL := FALSE;				//Ist das Licht invertiert? (NC)
	bAllFlanks		:	BOOL := FALSE;				//Alle Flanken verwenden?
	bSunIsDown		:	BOOL;
END_VAR
VAR_IN_OUT
	bInputHA		:	BOOL;						//Input (HA)
END_VAR
VAR_OUTPUT
	bOut			:	BOOL;
END_VAR
VAR CONSTANT
	nSize 			:	UINT := 5; 					//Maximale Anzahl Eingänge
END_VAR
VAR
	fbRtrig			:	ARRAY[0..nSize] OF R_TRIG;
	fbRtrigDoor		:	ARRAY[0..nSize] OF R_TRIG;
	fbFtrig			:	ARRAY[0..nSize] OF F_TRIG;
	Idx				:	UINT;
	bTrigger		:	BOOL;
END_VAR


IF bInputSec THEN	//Dauerlicht bei Security Falls
	
	IF bLightInv_NC THEN
		bOut		:= FALSE;
		bInputHA	:= TRUE;
	ELSE
		bOut		:= TRUE;
		bInputHA	:= TRUE;
	END_IF
	
ELSE	//Normale Funktion
	bTrigger := FALSE;

	//Init alle Flankentrigger und Frage diese ab
	FOR Idx := 0 TO nSize DO
	
		//Alle R_Trig
		fbRtrig[Idx](CLK:= bInputs[Idx], Q=> );
		fbRtrigDoor[Idx](CLK:= bInputsDoors[Idx], Q=> );
		
		bTrigger := bTrigger OR fbRtrig[Idx].Q;
	
		IF bAllFlanks THEN //Wenn alle Flanken
			fbFtrig[Idx](CLK:= bInputs[Idx], Q=> );
			bTrigger := bTrigger OR fbFtrig[Idx].Q;
		END_IF
	
		IF bSunIsDown THEN
			IF (NOT bOut AND NOT bLightInv_NC) OR (bOut AND bLightInv_NC) THEN 
				bTrigger := bTrigger OR fbRtrigDoor[Idx].Q;
			END_IF
		END_IF
		
	END_FOR
	

	IF bLightInv_NC THEN	//Wenn Licht Invertiert
	
		IF bInputHA THEN
			bOut	:= FALSE;
		ELSE
			bOut	:= TRUE;
		END_IF

	ELSE					//Wenn Licht nicht Invertiert 
		IF bInputHA THEN
			bOut	:= TRUE;
		ELSE
			bOut	:= FALSE;
		END_IF

	END_IF

	IF bTrigger THEN //Wenn Flanke erkannt
		bOut 			:= NOT bOut;
	
		IF bLightInv_NC THEN
			bInputHA	:= NOT bOut;
		ELSE
			bInputHa	:= bOut;
		END_IF
	END_IF
END_IF

END_FUNCTION_BLOCK

// ---- POUs/FB/FB_LightDimm.TcPOU
FUNCTION_BLOCK FB_LightDimm
VAR_INPUT
	bInputs				:	ARRAY[0..nSize] OF BOOL;	//Input Schalter oder Taster
	bInputSec			:	BOOL := FALSE;				//Input für Security Schaltung
	bInputSecTest		:	BOOL := FALSE;				//Testeingang für den Sec Modus
	bAllFlanks			:	BOOL := FALSE;				//Alle Flanken verwenden?
	bOnlyAtNight		:	BOOL := FALSE;				//Schalter funktioniert nur Nachts
	tLongPress			:	TIME := T#1000MS;			//Long Press Zeit für AUS!
	iNumPress4Dimm		:	UINT := 4;					//Reduktion der Helligkeit je Tastendruck
END_VAR
VAR_IN_OUT
	bInputHA		:	BOOL;						//Input (HA)
	iDimmValue		:	WORD;						//DimmValue Input
END_VAR
VAR_OUTPUT
	iOut			:	INT;
END_VAR
VAR CONSTANT
	nSize 			:	UINT := 5; 					//Maximale Anzahl Eingänge
END_VAR
VAR
	fbRtrig			:	ARRAY[0..nSize] OF R_TRIG;
	fbFtrig			:	ARRAY[0..nSize] OF F_TRIG;
	tonLongPress	:	ARRAY[0..nSize] OF TON;
	
	Idx				:	UINT;
	
	bSecRising		:	BOOL := TRUE;

END_VAR
VAR_TEMP
	iCountDimm		:	UINT;
	iCalcReduction	:	INT;
	
	bTrigger		:	BOOL := FALSE;
	bAllOFF			:	BOOL := FALSE;
END_VAR


IF bInputSec OR bInputSecTest THEN	//Party bei Security Falls
	
	bInputHA	:= TRUE;
	
	IF bSecRising THEN
		
		iDimmValue := iDimmValue + 5;

		IF iDimmValue = 255 THEN
			bSecRising := FALSE;
		END_IF	
	
	ELSE
	
		iDimmValue := iDimmValue - 5;

		IF iDimmValue <= 0 THEN
			bSecRising := TRUE;
		END_IF	
	
	END_IF

	
ELSE	//Normale Funktion

	//Init alle Flankentrigger und Frage diese ab
	FOR Idx := 0 TO nSize DO
	
		//Alle R_Trig
		fbRtrig[Idx](CLK:= bInputs[Idx], Q=> );
		tonLongPress[Idx](IN := bInputs[Idx], PT := tLongPress);
		
		bTrigger := bTrigger OR fbRtrig[Idx].Q;
		bAllOFF	:= bAllOFF OR tonLongPress[Idx].Q;
	
		IF bAllFlanks THEN //Wenn alle Flanken
			fbFtrig[Idx](CLK:= bInputs[Idx], Q=> );
			bTrigger := bTrigger OR fbFtrig[Idx].Q;
		END_IF
	
	END_FOR

	IF (iDimmValue > 0 OR bInputHA) AND iOut = 0 THEN		//Wenn über HA Eingeschaltet
		bInputHA	:= TRUE;
		
		IF iDimmValue = 0 THEN
			iDimmValue	:= 255;
		END_IF
	END_IF
	
	IF bOnlyAtNight THEN
		IF NOT gvl_mb.Output_Coils[19] THEN
			bTrigger	:= FALSE;
		END_IF
	END_IF
	
	IF bTrigger THEN
		
		IF iOut = 0 THEN					//Erstes Einschalten über Schalter
			bInputHA	:= TRUE;
			iDimmValue	:= 255;
		
		ELSE
			
			FOR iCountDimm := 0 TO iNumPress4Dimm DO
			
			iCalcReduction := (256 - (iCountDimm * (256 / iNumPress4Dimm)));
		
			IF iDimmValue > iCalcReduction THEN
				iDimmValue := iCalcReduction;
				EXIT;
			END_IF
		
			END_FOR
		
		END_IF
		
	END_IF

END_IF

IF bAllOFF OR bInputHA = FALSE OR iDimmValue <= 0 THEN		//Alles Ausschalten
	bInputHA	:= FALSE;
	iDimmValue	:= 0;
END_IF

iOut := F_LightDimmingConvertForHA(iDimmValue);

END_FUNCTION_BLOCK

// ---- POUs/Light/F_LightDimmingConvertForHA.TcPOU
FUNCTION F_LightDimmingConvertForHA : INT
VAR_INPUT
	iHA_DimmingValue	: INT;
END_VAR
VAR
	iConvertedValue		: INT;
END_VAR

(*---------------------------------------------------------
Converts a Dimming Value of Home Assistant (0-255) into a compatible 
Value for the Analog Output for Dimming (1-10V)
0V are not allowed as an Output. Ther must be a minimum of 1V (Dec:)
0V  =    0
1V  =  3276
10V = 32767
---------------------------------------------------------*)
IF iHA_DimmingValue = 255 THEN
	iConvertedValue := 32767;
ELSIF iHA_DimmingValue = 0 THEN
	iConvertedValue	:= 0;
ELSE
	iConvertedValue := 3276 + (iHA_DimmingValue * 115);
END_IF

F_LightDimmingConvertForHA := iConvertedValue;

END_FUNCTION

// ---- POUs/FB/FB_LightDimmIndirectNC.TcPOU
FUNCTION_BLOCK FB_LightDimmIndirectNC
VAR_INPUT
	bInputs				:	ARRAY[0..nSize] OF BOOL;	//Input Schalter oder Taster
	bInputSec			:	BOOL := FALSE;				//Input für Security Schaltung
	bInputSecTest		:	BOOL := FALSE;				//Testeingang für den Sec Modus
	bAllFlanks			:	BOOL := FALSE;				//Alle Flanken verwenden?
	tLongPress			:	TIME := T#1000MS;			//Long Press Zeit für AUS!
	tBlockTime			:	TIME := T#2000MS;			//Zeit nach Ausschalten bis wiedereinschalten
	iNumPress4Dimm		:	UINT := 4;					//Reduktion der Helligkeit je Tastendruck
END_VAR
VAR_IN_OUT
	bInputHA		:	BOOL;						//Input (HA)
	iDimmValue		:	WORD;						//DimmValue Input
END_VAR
VAR_OUTPUT
	iOut			:	INT;
	bOut			:	BOOL;
END_VAR
VAR CONSTANT
	nSize 			:	UINT := 5; 					//Maximale Anzahl Eingänge
END_VAR
VAR
	fbRtrig			:	ARRAY[0..nSize] OF R_TRIG;
	fbFtrig			:	ARRAY[0..nSize] OF F_TRIG;
	tonLongPress	:	ARRAY[0..nSize] OF TON;
	tonBlock		:	TON;
	
	Idx				:	UINT;
	
	bSecRising		:	BOOL := TRUE;
	bBlock			:	BOOL := FALSE;

END_VAR
VAR_TEMP
	iCountDimm		:	UINT;
	iCalcReduction	:	INT;
	
	bTrigger		:	BOOL := FALSE;
	bAllOFF			:	BOOL := FALSE;
END_VAR


tonBlock(IN := bBlock, PT := tBlockTime);

IF tonBlock.Q THEN
	bBlock	:= FALSE;
END_IF

IF (bInputSec OR bInputSecTest) AND NOT bBlock THEN	//Party bei Security Falls
	
	bInputHA	:= TRUE;
	bOut		:= FALSE;		// !!! NC
	
	IF bSecRising THEN
		
		iDimmValue := iDimmValue + 5;

		IF iDimmValue = 255 THEN
			bSecRising := FALSE;
		END_IF	
	
	ELSE
	
		iDimmValue := iDimmValue - 5;

		IF iDimmValue <= 0 THEN
			bSecRising := TRUE;
		END_IF	
	
	END_IF

	
ELSE	//Normale Funktion

	//Init alle Flankentrigger und Frage diese ab
	FOR Idx := 0 TO nSize DO
	
		//Alle R_Trig
		fbRtrig[Idx](CLK:= bInputs[Idx], Q=> );
		tonLongPress[Idx](IN := bInputs[Idx], PT := tLongPress);
		
		bTrigger := bTrigger OR fbRtrig[Idx].Q;
		bAllOFF	:= bAllOFF OR tonLongPress[Idx].Q;
	
		IF bAllFlanks THEN //Wenn alle Flanken
			fbFtrig[Idx](CLK:= bInputs[Idx], Q=> );
			bTrigger := bTrigger OR fbFtrig[Idx].Q;
		END_IF
	
	END_FOR

	IF (iDimmValue > 0 OR bInputHA) AND iOut = 0 AND NOT bBlock THEN		//Wenn über HA Eingeschaltet
		bInputHA	:= TRUE;
		bOut		:= FALSE;		// !!! NC
		
		IF iDimmValue = 0 THEN
			iDimmValue	:= 255;
		END_IF
	END_IF
	
	IF bTrigger AND NOT bBlock THEN
		
		IF iOut = 0 THEN					//Erstes Einschalten über Schalter
			bInputHA	:= TRUE;
			bOut		:= FALSE;			// !!! NC
			iDimmValue	:= 255;
		
		ELSE
			
			FOR iCountDimm := 0 TO iNumPress4Dimm DO
			
			iCalcReduction := (256 - (iCountDimm * (256 / iNumPress4Dimm)));
		
			IF iDimmValue > iCalcReduction THEN
				iDimmValue := iCalcReduction;
				EXIT;
			END_IF
		
			END_FOR
		
		END_IF
		
	END_IF

END_IF

IF bAllOFF OR bInputHA = FALSE OR iDimmValue <= 0 THEN		//Alles Ausschalten
	bInputHA	:= FALSE;
	bOut		:= TRUE;			// !!! NC
	iDimmValue	:= 0;
	bBlock		:= TRUE;
END_IF

iOut := F_LightDimmingConvertForHA(iDimmValue);

END_FUNCTION_BLOCK

// ---- POUs/FB/FB_LightPIR.TcPOU
FUNCTION_BLOCK FB_LightPIR
VAR_INPUT
	bInputPIR		:	BOOL;						//Input des Bewegungsmelders
	bInputSecLoop	:	BOOL := FALSE;				//Input für Security Loop
	tHigh			:	TIME;						//Zeit (ms) für High
END_VAR
VAR_IN_OUT
	bInputHA		:	BOOL;						//Input (HA)
END_VAR
VAR_OUTPUT
	bOut			:	BOOL;
END_VAR
VAR CONSTANT
	tSec			:	TIME := T#1S;
END_VAR
VAR
	fbRtrigPIR		:	R_TRIG;
	fbTrigSec		:	R_TRIG;
	
	bStateOut		:	BOOL := FALSE;

	tpPulse			:	TP_RST;
	
	tpPulseSec		:	TP;
	tofDelaySec		:	TOF;
END_VAR

// Security Loop
fbTrigSec	(CLK:= bInputPIR, Q=> );

IF bInputSecLoop THEN
	
	tpPulseSec	(IN := bStateOut, PT := tSec);
    tofDelaySec	(IN := bStateOut, PT := tSec);

	IF fbTrigSec.Q THEN
		bStateOut	:= TRUE;
	END_IF
	
	IF NOT tpPulseSec.Q THEN
		bStateOut := FALSE;
	END_IF
	
	IF NOT tofDelaySec.Q THEN
		bStateOut := TRUE;
	END_IF	

ELSIF bInputHA THEN

	bStateOut := TRUE;

ELSE

	fbRtrigPIR(CLK:= bInputPIR, Q=> );
	
	// Pulse
	tpPulse(IN := fbRtrigPIR.Q, PT := tHigh);

	IF tpPulse.Q THEN
		bStateOut	:= TRUE;
		
		//Reset Pulse bei neuer erkennung
		tpPulse.RST := fbRtrigPIR.Q;
		
	ELSE
		bStateOut 	:= FALSE;
	END_IF
	
	IF bInputPIR THEN
		bStateOut	:= TRUE;
	END_IF

END_IF

bOut		:= bStateOut;

END_FUNCTION_BLOCK

// ---- POUs/FB/TP_RST.TcPOU
FUNCTION_BLOCK TP_RST
VAR_INPUT
   IN : BOOL;
   PT : TIME;
   RST : BOOL;
END_VAR
VAR_OUTPUT
   Q : BOOL;
   ET : TIME;
END_VAR
VAR CONSTANT
   INIT : INT := 0;
   RUN_PULSE : INT := 1;
   PULSE_DONE : INT := 2;
   RESET_TIME : INT := 3;
END_VAR
VAR
   Timer : TON;
   State : INT;
END_VAR

CASE State OF
   INIT://Make sure output and timer are off
      Timer(IN:=FALSE, PT:=PT, ET=>ET);
      Q := FALSE;
      //See if user wants to start pulse
      IF IN THEN
         State := RUN_PULSE;
      END_IF
      
   RUN_PULSE://Normal pulse (output is true)
      Timer(IN:=TRUE, PT:=PT, ET=>ET);
      Q := TRUE;
      //See if timer reset requested
      IF RST THEN
         State := RESET_TIME;
      END_IF
      //See if timer expired (this overrides RST signal if timer is already done)
      IF Timer.Q THEN
         State := PULSE_DONE;
      END_IF
   
   PULSE_DONE://Pulse is done - ignore RST input
      //Keep timer TRUE to maintain ET like normal TP
      Timer(IN:=TRUE, PT:=PT, ET=>ET);
      Q := FALSE;
      //See if user shuts off timer
      IF NOT IN THEN
         State := INIT;
      END_IF
      
   RESET_TIME://User wants to extend pulse output (keep output high)
      //Reset timer (ET = 0 again)
      Timer(IN:=FALSE, PT:=PT, ET=>ET);
      Q := TRUE;
      //Watch for drop of RST - and go back to normal pulse output
      IF NOT RST THEN
         State := RUN_PULSE;
      END_IF
      
   ELSE //problem in code - reset state machine so FB doesn't freeze
      State := INIT;
      
END_CASE

END_FUNCTION_BLOCK

// ---- POUs/sub_Security.TcPOU
PROGRAM sub_Security
VAR

END_VAR

//###################################################################################
//##-----------------------------------SECURITY------------------------------------##
//###################################################################################

//--------------------Variablen Setzen----------------------------------
//ALARM GESAMT
IF gvl_mb.Output_Coils[240] THEN
	gvl_mb.Output_Coils[241] 	:= TRUE;
	gvl_mb.Output_Coils[244]	:= TRUE;
END_IF

//ALARM LICHT
IF gvl_mb.Output_Coils[241] THEN
	gvl_mb.Output_Coils[242]	:= TRUE;
	gvl_mb.Output_Coils[243]	:= TRUE;
END_IF

//ALARM NOIS
IF gvl_mb.Output_Coils[244] THEN
	gvl_mb.Output_Coils[245]	:= TRUE;
	gvl_mb.Output_Coils[246]	:= TRUE;
END_IF


//--------------------------------- INVERT Input Windows / Doors ------------------------
gvl_mb.Output_Coils[200] := NOT gvl_EA.bID24_01_3;		// Fensterkontakt Bad EG
gvl_mb.Output_Coils[201] := NOT gvl_EA.bID24_01_4;		// Fensterkontakt Büro
gvl_mb.Output_Coils[203] := NOT gvl_EA.bID24_02_1;		// Fensterkontakt Keller
gvl_mb.Output_Coils[204] := NOT gvl_EA.bID24_02_2;		// Fensterkontakt Technik
gvl_mb.Output_Coils[205] := NOT gvl_EA.bID24_02_3;		// Fensterkontakt Hobbyraum Süd
gvl_mb.Output_Coils[207] := NOT gvl_EA.bID24_02_4;		// Kontakt Terassentür UG
gvl_mb.Output_Coils[206] := NOT gvl_EA.bID24_03_1;		// Fensterkontakt Hobbyraum West
gvl_mb.Output_Coils[202] := NOT gvl_EA.bID24_03_2;		// Kontakt Balkontür
gvl_mb.Output_Coils[209] := NOT gvl_EA.bWID01_3;		// Reedkontakt Werkstatttür
gvl_mb.Output_Coils[208] := NOT gvl_EA.bWID01_4;		// Reedkontakt Werkstattfenster
gvl_mb.Output_coils[210] :=	NOT gvl_EA.bWID01_11; 		// TüR		OG	Garage Strasse
gvl_mb.Output_coils[211] :=	NOT gvl_EA.bWID01_12; 		// Fenster	OG	Garage
gvl_mb.Output_Coils[212] :=	NOT gvl_EA.bWID01_13; 		// TüR		OG	Garage Haus

gvl_mb.Output_coils[213] :=	gvl_EA.bWID01_15; 			// Garagentor offen
gvl_mb.Output_coils[214] := gvl_EA.bWID01_16; 			// Garagentor geschlossen
gvl_mb.Output_Coils[215] := gvl_EA.bWID01_14; 			// Garagentor Lüftung

END_PROGRAM

// ---- POUs/sub_Access.TcPOU
PROGRAM sub_Access
VAR
	
	bGarageStellungLueften	    : BOOL;
	bGarageStellungLueftenTemp	: BOOL;

	fbTuerGong			:	FB_Impulse;
	fbGaragentorToggle	:	FB_Impulse_LongPress;
	fbGaragentorAuf		:	FB_Impulse;
	fbGaragentorAb		:	FB_Impulse;
	fbGaragentorHalb	:	FB_Impulse;
	fbGaragentorLueften	:	FB_Impulse;
	fbgaragentorStatus	:	FB_GarageStatus;
	
	fbTuerGarageHaus	:	FB_Door;
	fbTuerGarageStrasse	:	FB_Door;
	fbTuerWerkstatt		:	FB_Door;
	fbTuerHaus			:	FB_Door;
	
END_VAR

//###################################################################################
//##-----------------------------------ACCESS--------------------------------------##
//###################################################################################

bGarageStellungLueften := FALSE;

//--------------------TürGong----------------------------------
fbTuerGong.bInputs[0]	:= gvl_EA.bID24_01_1;

fbTuerGong(
	bR_Trig			:= TRUE,
	bInputSecLoop	:= gvl_mb.Output_Coils[245],
	bInputHA		:= gvl_mb.Output_Coils[14],
	tHigh			:= T#500MS,
	bOut			=> gvl_EA.bOD02_3
);
//-------------------------------------------------------------

//--------------------Garagentor Stellung Auf----------------------------------
fbGaragentorAuf(
	bR_Trig			:= TRUE,
	bInputHA		:= gvl_mb.Output_Coils[38],
	tHigh			:= T#500MS,
	bOut			=> gvl_EA.bWOD01_14
);
//-------------------------------------------------------------

//--------------------Garagentor Stellung Ab----------------------------------
fbGaragentorAb(
	bR_Trig			:= TRUE,
	bInputHA		:= gvl_mb.Output_Coils[39],
	tHigh			:= T#500MS,
	bOut			=> gvl_EA.bWOD01_15
);
//-------------------------------------------------------------

//--------------------Garagentor Stellung Halb----------------------------------
fbGaragentorHalb(
	bR_Trig			:= TRUE,
	bInputHA		:= gvl_mb.Output_Coils[40],
	tHigh			:= T#500MS,
	bOut			=> gvl_EA.bWOD01_16
);
//-------------------------------------------------------------

//--------------------Garagentor Stellung Lüften----------------------------------
fbGaragentorLueften(
	bR_Trig			:= TRUE,
	bInputHA		:= gvl_mb.Output_Coils[37],
	tHigh			:= T#500MS,
	bOut			=> bGarageStellungLueftenTemp
);

bGarageStellungLueften := bGarageStellungLueften OR bGarageStellungLueftenTemp; 
//-------------------------------------------------------------

//--------------------Garagentor Stellung Toggle----------------------------------
fbGaragentorToggle(
	bInput			:= gvl_EA.bID05_1,
	bInputHA		:= gvl_mb.Output_Coils[13],
	tHigh			:= T#500MS,
	tLongPress		:= T#1S,
	bOut			=> gvl_EA.bWOD01_6,
	bOutLong		=> bGarageStellungLueftenTemp
);

bGarageStellungLueften := bGarageStellungLueften OR bGarageStellungLueftenTemp; 
//-------------------------------------------------------------

//--------------------Garagentor Status----------------------------------
fbGaragentorStatus(
	bInputOpened	:= gvl_EA.bWID01_15,
	bInputClosed	:= gvl_EA.bWID01_16,
	bInputAir		:= gvl_EA.bWID01_14,
	iOut			=> gvl_mb.Output_Registers[25]
);
//-------------------------------------------------------------

//--------------------Türöffner Garagentür Haus----------------------------------
fbTuerGarageHaus(
	bInput			:= gvl_EA.bWID01_9,
	bInputSwitch	:= gvl_EA.bID05_2,
	bInputHA		:= gvl_mb.Output_Coils[35],
	tPulse			:= T#3S,
	tPulseSwitch	:= T#10S,
	bOut			=> gvl_EA.bWOD01_11
);
//-------------------------------------------------------------

//--------------------Türöffner Garagentür Strasse----------------------------------
fbTuerGarageStrasse(
	bInput			:= gvl_EA.bWID01_8,
	bInputHA		:= gvl_mb.Output_Coils[34],
	tPulse			:= T#3S,
	bOut			=> gvl_EA.bWOD01_10
);
//-------------------------------------------------------------

//--------------------Türöffner Werkstatt----------------------------------
fbTuerWerkstatt(
	bInput			:= gvl_EA.bWID01_10,
	bInputHA		:= gvl_mb.Output_Coils[41],
	tPulse			:= T#3S,
	bOut			=> gvl_EA.bWOD02_1
);
//-------------------------------------------------------------

//--------------------Türöffner Haustür----------------------------------
fbTuerHaus(
	bInput			:= gvl_EA.bID24_01_2,
	bInputHA		:= gvl_mb.Output_Coils[16],
	bInputPerm		:= gvl_mb.Output_Coils[17],
	tPulse			:= T#5S,
	bOut			=> gvl_EA.bOD04_5
);
//-------------------------------------------------------------


gvl_EA.bWOD01_13 := bGarageStellungLueften;

END_PROGRAM

// ---- POUs/FB/FB_Impulse.TcPOU
FUNCTION_BLOCK FB_Impulse
VAR_INPUT
	bInputs			:	ARRAY[0..nSize] OF BOOL;	//Input Schalter oder Taster
	bInputSecLoop	:	BOOL := FALSE;				//Input für Security Loop
	bR_Trig			:	BOOL := TRUE;				//Steigende Flanke? Wenn FALSE = Fallend
	tHigh			:	TIME;						//Zeit (ms) für High
	tDelay			:	TIME := T#0MS;				//Verzögerungszeit (ms) zwischen den Impulsen									
END_VAR
VAR_OUTPUT
	bOut			:	BOOL;
END_VAR
VAR_IN_OUT
	bInputHA		:	BOOL;
END_VAR
VAR CONSTANT
	nSize 			:	UINT := 5; 					//Maximale Anzahl Eingänge
END_VAR
VAR
	fbRtrig			:	ARRAY[0..nSize] OF R_TRIG;
	fbFtrig			:	ARRAY[0..nSize] OF F_TRIG;
	
	fbRtrigInit		:	R_TRIG;
	
	Idx				:	UINT;
	bTrigger		:	BOOL;
	
	tpPulse			:	TP;
	tofDelay		:	TOF;
	
END_VAR
VAR_TEMP

END_VAR



//--------------------------------------Notfall Toggle
fbRtrigInit(CLK:= bInputSecLoop, Q=> );
tpPulse(IN := bOut, PT := tHigh);
tofDelay(IN := bOut, PT := tHigh);

IF bInputSecLoop THEN
		
	IF fbRtrigInit.Q THEN
		bOut	:= TRUE;
	END_IF
	
	IF NOT tpPulse.Q THEN
		bOut := FALSE;
	END_IF
	
	IF NOT tofDelay.Q THEN
		bOut := TRUE;
	END_IF	
	
ELSE //----------------------------------Normaler Impuls
	bTrigger 	:= FALSE;

	//Init alle Flankentrigger und Frage diese ab
	FOR Idx := 0 TO nSize DO
	
		IF bR_Trig THEN
		
			fbRtrig[Idx](CLK:= bInputs[Idx], Q=> );
			bTrigger := bTrigger OR fbRtrig[Idx].Q;
	
		ELSE
	
			fbFtrig[Idx](CLK:= bInputs[Idx], Q=> );
			bTrigger := bTrigger OR fbFtrig[Idx].Q;
	
		END_IF
	
	END_FOR
	
	bTrigger := bTrigger OR bInputHA;
	
	IF NOT tofDelay.Q THEN
		tpPulse(IN := bTrigger, PT := tHigh);
	END_IF

	IF tpPulse.Q THEN
		bOut 		:= TRUE;
		bInputHA 	:= TRUE;
	ELSE
		bOut 		:= FALSE;
		bInputHA	:= FALSE;
		tofDelay(IN := bOut, PT := tDelay);
	END_IF
	
END_IF

END_FUNCTION_BLOCK

// ---- POUs/FB/FB_Impulse_LongPress.TcPOU
FUNCTION_BLOCK FB_Impulse_LongPress
VAR_INPUT
	bInput			:	BOOL;	//Input Schalter oder Taster
	tHigh			:	TIME;						//Zeit (ms) für High
	tLongPress		:	TIME;							
END_VAR
VAR_OUTPUT
	bOut			:	BOOL;
	bOutLong		:	BOOL;
END_VAR
VAR_IN_OUT
	bInputHA		:	BOOL;
END_VAR
VAR CONSTANT
END_VAR
VAR
	fbFtrig			:	F_TRIG;
	bTrigger		:	BOOL;
	bOutTrig		:	BOOL;
	
	tpPulse			:	TP;
	tonLongPress	:	TON;
	
END_VAR
VAR_TEMP

END_VAR


tpPulse		 (IN := bOutTrig, PT := tHigh);
tonLongPress (IN := bInput, PT := tLongPress);

bTrigger 	:= FALSE;
		
fbFtrig(CLK:= bInput, Q=> );

//Normale Tastendruck
bTrigger := bTrigger OR fbFtrig.Q;

//Signal über HA
bTrigger := bTrigger OR bInputHA;

//Wenn normaler Tastendruck und Impuls noch nicht abgelaufen
IF (tpPulse.Q AND NOT bInput) OR bTrigger THEN
	bOut 		:= TRUE;
	bInputHA	:= FALSE;
//Wenn langer Tastendruck
ELSIF tonLongPress.Q OR (tpPulse.Q AND bInput) THEN
	bOutLong	:= TRUE;

//Wenn nichts
ELSE
	bOut 		:= FALSE;
	bOutLong	:= FALSE;
	bInputHA	:= FALSE;
	
	bOutTrig	:= FALSE;
END_IF
	
bOutTrig := bOut OR bOutLong;

END_FUNCTION_BLOCK

// ---- POUs/FB/FB_GarageStatus.TcPOU
FUNCTION_BLOCK FB_GarageStatus
VAR_INPUT
	bInputOpened	:	BOOL;
	bInputClosed	:	BOOL;
	bInputAir		:	BOOL;

END_VAR
VAR_OUTPUT
	iOut			:	INT;
END_VAR
VAR_IN_OUT
END_VAR
VAR CONSTANT
END_VAR
VAR
	fbRtrig			:	R_TRIG;
	fbRtrigSwitch	:	R_TRIG;
	fbRtrigHA		:	R_TRIG;
	
	tpPulse			:	TP;
	tpPulseSwitch	:	TP;
		
	bTrigger		:	BOOL;
	

	
	bInputOpenedAND: INT;
END_VAR
VAR_TEMP

END_VAR


IF bInputOpened AND NOT bInputClosed AND NOT bInputAir THEN
	//Geöffnet
	iOut := 3;
ELSIF NOT bInputOpened AND bInputClosed AND NOT bInputAir THEN
	//Geschlossen
	iOut := 2;
ELSIF NOT bInputOpened AND NOT bInputClosed AND bInputAir THEN
	//Lüftungstellung
	iOut := 1;
ELSE
	// Teilgeöffnet
	iOut := 0;
END_IF

END_FUNCTION_BLOCK

// ---- POUs/FB/FB_Door.TcPOU
FUNCTION_BLOCK FB_Door
VAR_INPUT
	bInput			:	BOOL;	// Input über ein System
	bInputSwitch	:	BOOL;	// Input über einen Taster
	bInputPerm		:	BOOL;	// Input für dauerhaftes öffnen
	
	tPulse			:	TIME := T#5S;	//Zeit für High bei System oder HomeAssistant
	tPulseSwitch	:	TIME := tPulse;	//Zeit für High bei Schalter 
END_VAR
VAR_OUTPUT
	bOut			:	BOOL;
END_VAR
VAR_IN_OUT
	bInputHA		:	BOOL;	// Input über Home Assistant Taster
END_VAR
VAR CONSTANT
END_VAR
VAR
	fbRtrig			:	R_TRIG;
	fbRtrigSwitch	:	R_TRIG;
	fbRtrigHA		:	R_TRIG;
	
	tpPulse			:	TP;
	tpPulseSwitch	:	TP;
		
	bTrigger		:	BOOL;
	

	
END_VAR
VAR_TEMP

END_VAR

IF bInputPerm THEN
	
	bOut := TRUE;
	
ELSE

	bTrigger 	:= FALSE;

	fbRtrig(CLK:= bInput, Q=> );
	fbRtrigSwitch(CLK:= bInputSwitch, Q=> );
	fbRtrigHA(CLK:= bInputHA, Q=> );

	bTrigger := bTrigger OR fbRtrig.Q OR fbRtrigHA.Q;
	
	tpPulse(IN := bTrigger, PT := tPulse);
	tpPulseSwitch(IN := fbRtrigSwitch.Q, PT := tPulseSwitch);

	IF tpPulse.Q OR tpPulseSwitch.Q THEN
		bOut 		:= TRUE;
	ELSE
		bOut 		:= FALSE;
		bInputHA	:= FALSE;
	END_IF
	
END_IF

END_FUNCTION_BLOCK

// ---- POUs/sub_Power.TcPOU
PROGRAM sub_Power
VAR
		fbPowerWerkstatt		:	FB_PowerSocket;
		fbPowerFernseher		:	FB_PowerSocket;
		fbPowerUhr				:	FB_PowerSocket;
		fbPowerEsszimmer		:	FB_PowerSocket;
		fbPowerAussenHaustur	:	FB_PowerSocket;
		fbPowerAussenBalkon		:	FB_PowerSocket;
		fbPowerZisterne			:	FB_PowerSocket;
		fbPowerSmartMirror		:	FB_PowerSocket;
		fbPowerLEDBandWohn		:	FB_PowerSocket;
		fbPowerLadeWerkstatt	:	FB_PowerSocket;
		fbPowerLadeGarage		:	FB_PowerSocket;
		fbPowerGaragenDach		:	FB_PowerSocket;
		
END_VAR

//###################################################################################
//##-----------------------------------POWER---------------------------------------##
//###################################################################################

//--------------------WERKSTATT STECKDOSE----------------------------------
fbPowerWerkstatt.bInputs[0] 	:= gvl_EA.bWID01_2;

fbPowerWerkstatt
(
	bPowerInv_NC	:=	TRUE,
	bInputHA		:=	gvl_mb.Output_Coils[12]	,
	bOut			=>	gvl_EA.bWOD01_2,
);
//-------------------------------------------------------------------------

//--------------------FERNSEHER STECKDOSE----------------------------------
fbPowerFernseher
(
	bPowerInv_NC	:=	TRUE,
	bInputHA		:=	gvl_mb.Output_Coils[18],
	bOut			=>	gvl_EA.bOD02_6,
);
//-------------------------------------------------------------------------

//--------------------UHR STECKDOSE----------------------------------
fbPowerUhr
(
	bInputHA		:=	gvl_mb.Output_Coils[11],
	bOut			=>	gvl_EA.bOD02_5,
);
//-------------------------------------------------------------------------

//--------------------ESSZIMMER STECKDOSE----------------------------------
fbPowerEsszimmer
(
	bInputHA		:=	gvl_mb.Output_Coils[20],
	bOut			=>	gvl_EA.bOD02_4,
);
//-------------------------------------------------------------------------

//--------------------HAUSTÜR AUSSENSTECKDOSE----------------------------------
fbPowerAussenHaustur
(
	bInputHA		:=	gvl_mb.Output_Coils[21],
	bOut			=>	gvl_EA.bOD02_7,
);
//-------------------------------------------------------------------------

//--------------------BALKON AUSSENSTECKDOSE----------------------------------
fbPowerAussenBalkon
(
	bInputHA		:=	gvl_mb.Output_Coils[22],
	bOut			=>	gvl_EA.bOD02_8,
);
//-------------------------------------------------------------------------

//--------------------STROM ZISTERNE----------------------------------
fbPowerZisterne
(
	bInputHA		:=	gvl_mb.Output_Coils[23],
	bOut			=>	gvl_EA.bOD03_6,
);
//-------------------------------------------------------------------------

//--------------------STROM SMARTMIRROR----------------------------------
fbPowerSmartMirror
(
	bInputHA		:=	gvl_mb.Output_Coils[24],
	bOut			=>	gvl_EA.bOD04_2,
);
//-------------------------------------------------------------------------

//--------------------LED-BAND WOHNZIMMER STECKDOSE-------------------------------
fbPowerLEDBandWohn
(
	bInputHA		:=	gvl_mb.Output_Coils[25],
	bOut			=>	gvl_EA.bOD04_3,
);
//-------------------------------------------------------------------------

//--------------------LADEGERÄTE WERKSTATT----------------------------------
fbPowerLadeWerkstatt
(
	bInputHA		:=	gvl_mb.Output_Coils[27],
	bOut			=>	gvl_EA.bWOD01_5,
);
//-------------------------------------------------------------------------

//--------------------LADEGERÄTE GARAGE----------------------------------
fbPowerLadeGarage
(
	bInputHA		:=	gvl_mb.Output_Coils[43],
	bOut			=>	gvl_EA.bWOD02_2,
);
//-------------------------------------------------------------------------

//--------------------STECKDOSE GARAGENDACH----------------------------------
fbPowerGaragenDach
(
	bInputHA		:=	gvl_mb.Output_Coils[44],
	bOut			=>	gvl_EA.bWOD02_3,
);
//-------------------------------------------------------------------------

END_PROGRAM

// ---- POUs/FB/FB_PowerSocket.TcPOU
FUNCTION_BLOCK FB_PowerSocket
VAR_INPUT
	bInputs			:	ARRAY[0..nSize] OF BOOL;	//Input Schalter oder Taster
	bPowerInv_NC	:	BOOL := FALSE;				//Ist die Schaltung invertiert? (NC)
	bAllFlanks		:	BOOL := FALSE;				//Alle Flanken verwenden?
END_VAR
VAR_IN_OUT
	bInputHA		:	BOOL;						//Input (HA)
END_VAR
VAR_OUTPUT
	bOut			:	BOOL;
END_VAR
VAR CONSTANT
	nSize 			:	UINT := 5; 					//Maximale Anzahl Eingänge
END_VAR
VAR
	fbRtrig			:	ARRAY[0..nSize] OF R_TRIG;
	fbFtrig			:	ARRAY[0..nSize] OF F_TRIG;
	Idx				:	UINT;
	bTrigger		:	BOOL;
END_VAR


bTrigger := FALSE;

//Init alle Flankentrigger und Frage diese ab
FOR Idx := 0 TO nSize DO
	
	//Alle R_Trig
	fbRtrig[Idx](CLK:= bInputs[Idx], Q=> );
	bTrigger := bTrigger OR fbRtrig[Idx].Q;
	
	IF bAllFlanks THEN //Wenn alle Flanken
		fbFtrig[Idx](CLK:= bInputs[Idx], Q=> );
		bTrigger := bTrigger OR fbFtrig[Idx].Q;
	END_IF
	
END_FOR

IF bPowerInv_NC THEN	//Wenn Schaltung Invertiert
	
	IF bInputHA THEN
		bOut	:= FALSE;
	ELSE
		bOut	:= TRUE;
	END_IF

ELSE					//Wenn Licht nicht Invertiert 
	IF bInputHA THEN
		bOut	:= TRUE;
	ELSE
		bOut	:= FALSE;
	END_IF

END_IF

IF bTrigger THEN //Wenn Flanke erkannt
	
	bOut 			:= NOT bOut;
	
	IF bPowerInv_NC THEN
		bInputHA	:= NOT bOut;
	ELSE
		bInputHa	:= bOut;
	END_IF

END_IF

END_FUNCTION_BLOCK

// ---- POUs/sub_Measure.TcPOU
PROGRAM sub_Measure
VAR
		fbWaterConsumption			:	FB_Count;
		fbWaterConsumptionZisterne	:	FB_Count;
		fbWaterRain					:	FB_Count;
		
		fbHumWohnzimmer		:	FB_Con_2_Value;
		fbHumTechnikraum	:	FB_Con_2_Value;
		fbHumWerkstatt		:	FB_Con_2_Value;
		fbHumGarage			:	FB_Con_2_Value;
		
		fbCO2Wohnzimmer		:	FB_Convert_2co2;
		
		fbZisterne			:	FB_Convert_2Zisterne;
		
		fbTempGarage		:	FB_Convert_2temp;
		fbTempWerkstatt		:	FB_Convert_2temp;
		fbTempTechnikraum	:	FB_Convert_2temp;
		fbTempWohnzimmer	:	FB_Convert_2temp;
		
		
		//-----------AUSSEN------------------------
		fbWetterWindspeed	:	FB_Con_2_Value;
		fbWetterWindDir		:	FB_Con_2_Value;
		fbWetterLUX			:	FB_Con_2_Value;
		fbWetterTemp		:	FB_Con_2_Value;
		fbWetterHum			:	FB_Con_2_Value;

END_VAR

//###################################################################################
//##-----------------------------------MEASUREMENT---------------------------------##
//###################################################################################


gvl_mb.Output_Registers[19] := INT_TO_WORD(gvl_EA.iIAPT_01_1);	// Temperatur Bühne

//--------------------WATER CONSUMPTION Trinkwasser (1 = 10 Liter)-------------------
fbWaterConsumption
(
	bInput			:= gvl_EA.bID24_03_3,
	bAllFlanks 		:= FALSE,
	wCountRetain	:= gvl_RETAIN.waterConsumption,
	wOut			=> gvl_mb.Output_Registers[0]
);
//-----------------------------------------------------------------------
//--------------------WATER CONSUMPTION Zisterne (1 = 1 Liter)-------------------
fbWaterConsumptionZisterne
(
	bInput			:= gvl_EA.bID24_03_4,
	bAllFlanks 		:= FALSE,
	wCountRetain	:= gvl_RETAIN.waterConsumptionZisterne,
	wOut			=> gvl_mb.Output_Registers[22]
);
//-----------------------------------------------------------------------
//--------------------HUMIDITY WOHNZIMMER--------------------------------
fbHumWohnzimmer
(
	iInput			:= gvl_EA.iIAV01_2,
	tRefresh 		:= T#120S,
	diUppMeasureVal	:= 100,
	diLowMeasureVal	:= 0,
	wOut	 		=> gvl_mb.Output_Registers[15]
);
//-----------------------------------------------------------------------
//--------------------HUMIDITY TECHNIKRAUM--------------------------------
fbHumTechnikraum
(
	iInput			:= gvl_EA.iIAV02_1,
	tRefresh 		:= T#120S,
	diUppMeasureVal	:= 100,
	diLowMeasureVal	:= 0,
	wOut	 		=> gvl_mb.Output_Registers[18]
);
//-----------------------------------------------------------------------
//--------------------HUMIDITY WERKSTATT--------------------------------
fbHumWerkstatt
(
	iInput			:= gvl_EA.iWIAV01_2,
	tRefresh 		:= T#120S,
	diUppMeasureVal	:= 100,
	diLowMeasureVal	:= 0,
	wOut	 		=> gvl_mb.Output_Registers[21]
);
//-----------------------------------------------------------------------
//--------------------HUMIDITY GARAGE--------------------------------
fbHumGarage
(
	iInput			:= gvl_EA.iWIAV01_3,
	tRefresh 		:= T#120S,
	diUppMeasureVal	:= 100,
	diLowMeasureVal	:= 0,
	wOut	 		=> gvl_mb.Output_Registers[24]
);
//-----------------------------------------------------------------------
//--------------------WETTER HUMIDITY--------------------------------
fbWetterHum
(
	iInput			:= gvl_EA.iWIAA01_1,
	tRefresh 		:= T#120S,
	diUppMeasureVal	:= 100,
	diLowMeasureVal	:= 0,
	diOut	 		=> gvl_ha.diWetterHUM
);
//-----------------------------------------------------------------------
//--------------------CO2 WOHNZIMMER-------------------------------------
fbCO2Wohnzimmer
(
	iInput		:= gvl_EA.iIAV01_3,
	tRefresh 	:= T#120S,
	wOut 		=> gvl_mb.Output_Registers[16]
);
//-----------------------------------------------------------------------
//--------------------TEMP GARAGE-------------------------------------
fbTempGarage
(
	iInput		:= gvl_EA.iWIAV01_4,
	tRefresh 	:= T#120S,
	itempMAX	:= 70,
	itempMIN	:= -30,
	wOut 		=> gvl_mb.Output_Registers[23]
);
//-----------------------------------------------------------------------
//--------------------TEMP WERKSTATT-------------------------------------
fbTempWerkstatt
(
	iInput		:= gvl_EA.iWIAV01_1,
	tRefresh 	:= T#120S,
	itempMAX	:= 70,
	itempMIN	:= -30,
	wOut 		=> gvl_mb.Output_Registers[20]
);
//-----------------------------------------------------------------------
//--------------------TEMP TECHNIKRAUM-------------------------------------
fbTempTechnikraum
(
	iInput		:= gvl_EA.iIAV01_4,
	tRefresh 	:= T#120S,
	itempMAX	:= 70,
	itempMIN	:= -30,
	wOut 		=> gvl_mb.Output_Registers[17]
);
//-----------------------------------------------------------------------
//--------------------TEMP WOHNZIMMER-------------------------------------
fbTempWohnzimmer
(
	iInput		:= gvl_EA.iIAV01_1,
	tRefresh 	:= T#120S,
	itempMAX	:= 50,
	itempMIN	:= 0,
	wOut 		=> gvl_mb.Output_Registers[14]
);
//-----------------------------------------------------------------------
//--------------------WETTER TEMP-------------------------------------
fbWetterTemp
(
	iInput			:= gvl_EA.iWIAA01_2,
	tRefresh 		:= T#120S,
	diUppMeasureVal	:= 70,
	diLowMeasureVal	:= -30,
	iResultMulti	:= 10,
	diOut	 		=> gvl_ha.diWetterTEMP
);
//-----------------------------------------------------------------------
//--------------------ZISTERNE-------------------------------------
fbZisterne
(
	iInput		:= gvl_EA.iIAA01_1,
	tRefresh 	:= T#120S,
	wOutPerc	=> gvl_mb.Output_Registers[12],
	wOutLiter	=> gvl_mb.Output_Registers[13]

);
//-----------------------------------------------------------------------
//--------------------WETTER WINDSPEED--------------------------------
fbWetterWindspeed
(
	iInput			:= gvl_EA.iWIAA02_1,
	tRefresh 		:= T#1S,
	diUppMeasureVal	:= 35,
	diLowMeasureVal	:= 0,
	iResultMulti	:= 36,	//*3,6 (kmh) *10 komma Shift
	diOut	 		=> gvl_ha.diWetterWINDspeed
);
//-----------------------------------------------------------------------
//--------------------WETTER WIND DIRECTION--------------------------------
fbWetterWindDir
(
	iInput			:= gvl_EA.iWIAA02_2,
	tRefresh 		:= T#1S,
	diUppMeasureVal	:= 360,
	diLowMeasureVal	:= 0,
	diOut	 		=> gvl_ha.diWetterWINDdir
);
//-----------------------------------------------------------------------
//--------------------WATER Regenmenge (1 = 0.3mm)-------------------
fbWaterRain
(
	bInput			:= gvl_EA.bWID02_2,
	bAllFlanks 		:= FALSE,
	rMultiplier		:= 0.3,
	iFactor			:= 10,
	wCountRetain	:= gvl_RETAIN.waterRain,
	wOut			=> gvl_ha.wWetterRAIN
);

gvl_ha.bWetterRAIN := gvl_ea.bWID02_3;
//-----------------------------------------------------------------------
//--------------------WETTER LUX--------------------------------
fbWetterLUX
(
	iInput			:= gvl_EA.iWIAA02_3,
	tRefresh 		:= T#10S,
	diUppMeasureVal	:= 100000,
	diLowMeasureVal	:= 0,
	diOut	 		=> gvl_ha.diWetterLUX
);
//-----------------------------------------------------------------------

END_PROGRAM

// ---- POUs/FB/FB_Count.TcPOU
FUNCTION_BLOCK FB_Count
VAR_INPUT
	bInput				:	BOOL;	
	bAllFlanks			:	BOOL := FALSE;				//Alle Flanken verwenden?
	rMultiplier			:	REAL := 1;					//Wert wirt mit wOut multipliziert
	iFactor				:	INT	:= 1;					//Factor to shift komma
END_VAR
VAR_OUTPUT
	wOut				:	WORD;
END_VAR
VAR_IN_OUT
	wCountRetain		:	WORD;
END_VAR
VAR
	fbRTrig				:	R_TRIG;
	fbFTrig				:	F_TRIG;
	
	iMaxValue			:	UINT := 65535;
END_VAR


fbRTrig(CLK:= bInput, Q=> );

IF fbRTrig.Q THEN
	wCountRetain := TO_WORD((wCountRetain + 1) MOD REAL_TO_UINT(iMaxValue / (rMultiplier * iFactor)));
END_IF	

IF bAllFlanks THEN
	fbFTrig(CLK:= bInput, Q=> );

	IF fbFTrig.Q THEN
		wCountRetain := TO_WORD((wCountRetain + 1) MOD REAL_TO_UINT(iMaxValue / (rMultiplier * iFactor)));
	END_IF	
END_IF
	
wOut	:= REAL_TO_WORD((wCountRetain * rMultiplier)*iFactor);

END_FUNCTION_BLOCK

// ---- POUs/FB/FB_Con_2_Value.TcPOU
FUNCTION_BLOCK FB_Con_2_Value
VAR_INPUT
	iInput			:	INT;
	
	tRefresh		:	TIME;
	
	diUpperMax		:	DINT	:= 32767;
	diLowerMin		:	DINT	:= 0;
	diUppMeasureVal	:	DINT;
	diLowMeasureVal	:	DINT;

	iResultMulti	:	INT		:= 1;
END_VAR
VAR_OUTPUT
	diOut			:	DINT;
	wOut			:	WORD;
END_VAR
VAR
	rX				:	REAL;
	tonBlock		:	TON;
	
	bInit			:	BOOL := FALSE;
	
	rValuePerStep	:	REAL;
END_VAR

//Blocker for refresh interval
tonBlock(IN := NOT tonBlock.Q, PT := tRefresh);

IF NOT bInit THEN
	//Calculate inital Step Size
	rValuePerStep	:= ( (DINT_TO_REAL(diUppMeasureVal + (diLowMeasureVal * (-1)))) / DINT_TO_REAL(32767));
	bInit := TRUE;
END_IF

IF tonBlock.Q THEN
	//Check for Value to set for Max Output
	IF (iInput < diLowerMin) THEN
		rX := DINT_TO_REAL(diLowMeasureVal);

	//Check for Value to set for Min Output
	ELSIF (iInput > diUpperMax) THEN
		rx := DINT_TO_REAL(diUppMeasureVal);

	//Regular calculation
	ELSE
		rX := iInput * rValuePerStep;
		
		//Reduce to minus value if needed
		IF diLowMeasureVal < 0 THEN
		
			rX := rX + DINT_TO_REAL(diLowMeasureVal);
			// plus bec. values is MNUS
		
		END_IF
	END_IF
	
	IF rX > DINT_TO_REAL(diUppMeasureVal) THEN
	
		rX := DINT_TO_REAL(diUppMeasureVal);
	
	ELSIF rX < DINT_TO_REAL(diLowMeasureVal) THEN
		
		rX := DINT_TO_REAL(diLowMeasureVal);
		
	END_IF
	
	diOut 	:= REAL_TO_DINT(rX * iResultMulti);
	wOut	:= REAL_TO_WORD(rX * iResultMulti);
	

	
END_IF

END_FUNCTION_BLOCK

// ---- POUs/FB/FB_Convert_2co2.TcPOU
FUNCTION_BLOCK FB_Convert_2co2
VAR_INPUT
	iInput			:	INT;
	tRefresh		:	TIME;
END_VAR
VAR_OUTPUT
	wOut			:	WORD;
END_VAR
VAR
	rX				:	REAL;
	tonBlock		:	TON;
END_VAR

// For Convertion of 0-10V Signal from 0-2000ppm
tonBlock(IN := NOT tonBlock.Q, PT := tRefresh);

IF tonBlock.Q THEN

	rX := iInput * 0.061037018951994; //Annahme 10V entspr. 32767
	wOut := REAL_TO_WORD(rX);
	
END_IF

END_FUNCTION_BLOCK

// ---- POUs/FB/FB_Convert_2Zisterne.TcPOU
FUNCTION_BLOCK FB_Convert_2Zisterne
VAR_INPUT
	iInput			:	INT;
	tRefresh		:	TIME;
END_VAR
VAR_OUTPUT
	wOutPerc		: WORD;
	wOutLiter		: WORD;
END_VAR
VAR
	iValueArith		: INT;
	iPercent		: REAL;
	iLiter			: REAL;
	tonBlock		: TON;
	fbArithMittel	: FB_ArithMittel10;
	i_finalValue	: INT;
	
	iMaxValofSensor : REAL := 20000;
	
	
END_VAR

tonBlock(IN := NOT tonBlock.Q, PT := tRefresh);

IF tonBlock.Q THEN
	
	fbArithMittel(iInputValue := iInput, iOut => iValueArith );
	
	//-------------------- Prozent ------------------------
	
	iPercent	:= (iValueArith / iMaxValofSensor) * 100;
	
	IF iPercent > 100 THEN
		iPercent := 100;
	END_IF
	
	//-----------------------------------------------------
	
	//-------------------- Liter --------------------------
	
	iLiter := (iPercent / 100) * 5000;
	
	//------------------------------------------------
	
	wOutPerc	:= REAL_TO_WORD(iPercent);
	wOutLiter	:= REAL_TO_WORD(iLiter);
	
END_IF

END_FUNCTION_BLOCK

// ---- POUs/FB/FB_ArithMittel10.TcPOU
FUNCTION_BLOCK FB_ArithMittel10
VAR_INPUT
	iInputValue	: INT;
END_VAR
VAR_OUTPUT
	iOut		: INT;
END_VAR
VAR
	value 		: ARRAY [0..9] OF INT;
	counter		: INT 	:= 0;
	counter2	: INT	:= 0;
	x			: REAL 	:= 0;
	bInit		: BOOL	:= FALSE;
END_VAR


value[counter]  := iInputValue;

//Initialisierung abgeschlossen
IF counter = 9 THEN
	bInit	:= TRUE;
END_IF

IF bInit THEN
	
	x := 0;

	// Berechnung
	FOR counter2 := 0 TO 9 BY 1 DO
    	x := x + value[counter2];
	END_FOR;
		
	x := x / 10;	//Mitteln
	
	iOut := REAL_TO_INT(x);
	
ELSE
	iOut := 0;
END_IF

counter := (counter + 1) MOD 10;

END_FUNCTION_BLOCK

// ---- POUs/FB/FB_Convert_2temp.TcPOU
FUNCTION_BLOCK FB_Convert_2temp
VAR_INPUT
	iInput			:	INT;
	tRefresh		:	TIME;
	itempMAX		:	INT;
	iTempMIN		:	INT;
END_VAR
VAR_OUTPUT
	wOut			:	WORD;
END_VAR
VAR
	rX				:	REAL;
	tonBlock		:	TON;
	
	rMaxTempStep	:	REAL;
	rValuePerStep	:	REAL;
	bInit			:	BOOL := FALSE;
	iOut			:	INT;
END_VAR

// For Convertion of 0-10V Signal from 0-100%
tonBlock(IN := NOT tonBlock.Q, PT := tRefresh);

IF NOT bInit THEN
	rMaxTempStep	:= INT_TO_REAL(iTempMax + (iTempMin * (-1)));
	rValuePerStep	:= (rMaxTempStep / INT_TO_REAL(32767));

	bInit := TRUE;
END_IF


IF tonBlock.Q THEN

	rX := INT_TO_REAL(iInput) * rValuePerStep;
	
	rX := rX + INT_TO_REAL(iTempMIN);

	
	iOut := REAL_TO_INT(rX * 10.0);
	wOut := INT_TO_WORD(iOut);
	
END_IF

END_FUNCTION_BLOCK

// ---- POUs/sub_Heating.TcPOU
PROGRAM sub_Heating
VAR
	fbVitramoBadOG		:	FB_Heating;
	
	fbFanGarage			:	FB_Fan;
	fbFanWerkstatt		:	FB_Fan;
END_VAR

//###################################################################################
//##-----------------------------------HEATING-------------------------------------##
//###################################################################################

//--------------------------------ENTFEUCHTER WERKSTATT------------------------
gvl_ea.bWOD01_3 := gvl_mb.Output_Coils[42];
//-----------------------------------------------------------------------------
//--------------------------------VITRAMO BAD----------------------------------
fbVitramoBadOG
(
	bInput			:=	gvl_EA.bID04_4,
	bInputOverwrite	:=	gvl_mb.Output_Coils[15],
	bOut			=>	gvl_EA.bOD04_4
);
//-----------------------------------------------------------------------------
//--------------------------------FAN Garage----------------------------------
fbFanGarage
(
	bInputControl	:=	gvl_EA.bWID01_14,
	bInputHA		:=	gvl_mb.Output_Coils[33],
	bOut			=>	gvl_EA.bWOD01_9,
	bOut			=>	gvl_mb.Output_Coils[33],
);
//-----------------------------------------------------------------------------
//--------------------------------FAN Werkstatt----------------------------------
fbFanWerkstatt
(
	bInputControl			:=	gvl_EA.bWID01_2,
	bLongPressControlled 	:=	TRUE,
	tLongPress				:=  T#1S,
	bInputHA				:=	gvl_mb.Output_Coils[26],
	bOut					=>	gvl_EA.bWOD01_4,
	bOut					=>	gvl_mb.Output_Coils[26],
);
//-----------------------------------------------------------------------------

END_PROGRAM

// ---- POUs/FB/FB_Heating.TcPOU
FUNCTION_BLOCK FB_Heating
VAR_INPUT
	bInput			:	BOOL;
	bInputOverwrite	:	BOOL;
END_VAR
VAR_OUTPUT
	bOut			:	BOOL;
END_VAR
VAR
END_VAR

IF bInputOverwrite THEN
	bOut := TRUE;
ELSE
	bOut := bInput;
END_IF

END_FUNCTION_BLOCK

// ---- POUs/FB/FB_Fan.TcPOU
FUNCTION_BLOCK FB_Fan
VAR_INPUT
	bInputControl			:	BOOL;
	tLongPress				:	TIME;
	bLongPressControlled	: 	BOOL	:= FALSE;
	bInputHA				:	BOOL;						//Input (HA)
END_VAR
VAR_IN_OUT
END_VAR
VAR_OUTPUT
	bOut			:	BOOL;
END_VAR
VAR CONSTANT
END_VAR
VAR
	tonLongPress	:	TON;
	fbRTrigLong		:	R_Trig;
	
	fbRTrigHA		:	R_TRIG;
	fbFTrigHA		:	F_TRIG;

	fbRTrigInput	:	R_TRIG;
	fbFTrigInput	:	F_TRIG;

END_VAR


fbRTrigHA(CLK:= bInputHA, Q=> );
fbFTrigHA(CLK:= bInputHA, Q=> );

fbRTrigInput(CLK:= bInputControl, Q=> );
fbFTrigInput(CLK:= bInputControl, Q=> );

IF bLongPressControlled THEN
	
	tonLongPress (IN := bInputControl, PT := tLongPress);
	fbRTrigLong(CLK:= tonLongPress.Q, Q=> );

	IF fbRTrigLong.Q THEN
		bOut 		:= 	NOT bOut;
	END_IF

ELSE

	IF fbRTrigInput.Q THEN
		bOut	:=	TRUE;
	END_IF

	IF fbFTrigInput.Q THEN
		bOUT	:=	FALSE;
	END_IF

END_IF

IF fbRTrigHA.Q THEN
	bOut	:=	TRUE;
END_IF

IF fbFTrigHA.Q THEN
	bOUT	:=	FALSE;
END_IF

END_FUNCTION_BLOCK

// ---- POUs/Light/F_DimmAlgoForSwitch.TcPOU
FUNCTION F_DimmAlgoForSwitch : INT
VAR_INPUT
	i_DimmingValue	: INT;
END_VAR
VAR_OUTPUT
	bTurnOffTheLight : BOOL := FALSE;
END_VAR
VAR
END_VAR

(*---------------------------------------------------------
Defines the Dimming Algorithm for dimmable Lights by standard switch
---------------------------------------------------------*)
IF i_DimmingValue > 192 THEN 	//Wenn Leuchtkraft > 75%
		i_DimmingValue := 192;
	ELSIF i_DimmingValue > 128 THEN //Wenn Leuchtkraft > 50%
		i_DimmingValue := 128;
	ELSIF i_DimmingValue > 64 THEN 	//Wenn Leuchtkraft > 25%
		i_DimmingValue := 64;
	ELSIF i_DimmingValue <= 64 THEN 	//Wenn Leuchtkraft bei 25%
		bTurnOffTheLight := TRUE;
	END_IF

F_DimmAlgoForSwitch := i_DimmingValue;

END_FUNCTION
